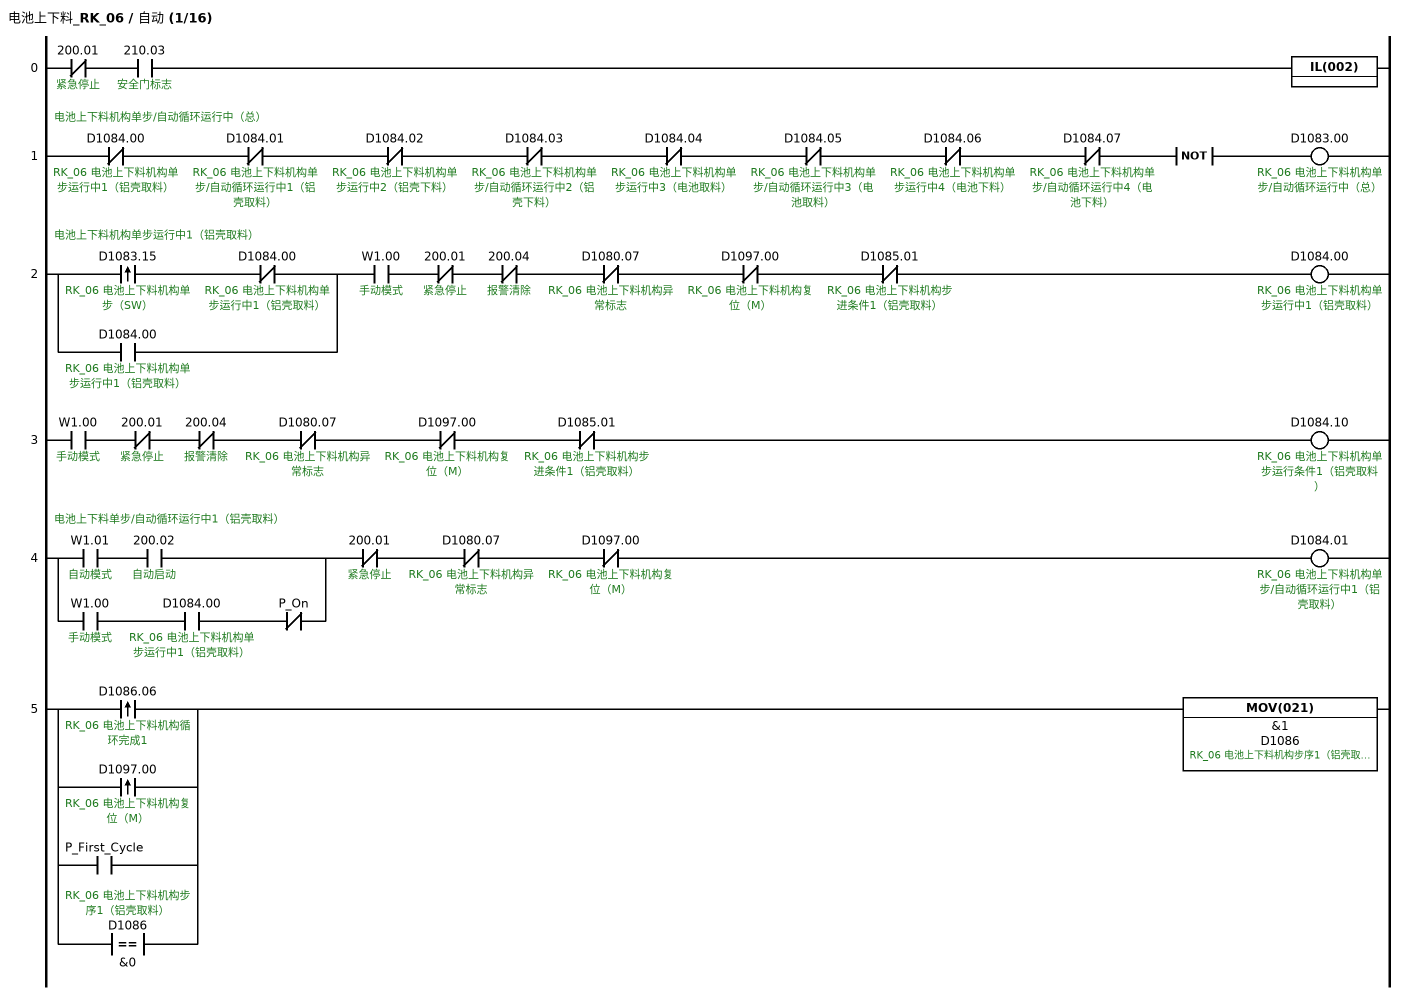
; [picture p528: 电池上下料_RK_06 / 自动, rungs 0-5]
; rung 0
LDNOT 200.01  ; 紧急停止
AND 210.03  ; 安全门标志
IL(002)
; rung 1: 电池上下料机构单步/自动循环运行中（总）
LDNOT D1084.00  ; RK_06 电池上下料机构单步运行中1（铝壳取料）
ANDNOT D1084.01  ; RK_06 电池上下料机构单步/自动循环运行中1（铝壳取料）
ANDNOT D1084.02  ; RK_06 电池上下料机构单步运行中2（铝壳下料）
ANDNOT D1084.03  ; RK_06 电池上下料机构单步/自动循环运行中2（铝壳下料）
ANDNOT D1084.04  ; RK_06 电池上下料机构单步运行中3（电池取料）
ANDNOT D1084.05  ; RK_06 电池上下料机构单步/自动循环运行中3（电池取料）
ANDNOT D1084.06  ; RK_06 电池上下料机构单步运行中4（电池下料）
ANDNOT D1084.07  ; RK_06 电池上下料机构单步/自动循环运行中4（电池下料）
NOT(520)
OUT D1083.00  ; RK_06 电池上下料机构单步/自动循环运行中（总）
; rung 2: 电池上下料机构单步运行中1（铝壳取料）
@LD D1083.15  ; RK_06 电池上下料机构单步（SW）
ANDNOT D1084.00  ; RK_06 电池上下料机构单步运行中1（铝壳取料）
OR D1084.00  ; RK_06 电池上下料机构单步运行中1（铝壳取料）
AND W1.00  ; 手动模式
ANDNOT 200.01  ; 紧急停止
ANDNOT 200.04  ; 报警清除
ANDNOT D1080.07  ; RK_06 电池上下料机构异常标志
ANDNOT D1097.00  ; RK_06 电池上下料机构复位（M）
ANDNOT D1085.01  ; RK_06 电池上下料机构步进条件1（铝壳取料）
OUT D1084.00  ; RK_06 电池上下料机构单步运行中1（铝壳取料）
; rung 3
LD W1.00  ; 手动模式
ANDNOT 200.01  ; 紧急停止
ANDNOT 200.04  ; 报警清除
ANDNOT D1080.07  ; RK_06 电池上下料机构异常标志
ANDNOT D1097.00  ; RK_06 电池上下料机构复位（M）
ANDNOT D1085.01  ; RK_06 电池上下料机构步进条件1（铝壳取料）
OUT D1084.10  ; RK_06 电池上下料机构单步运行条件1（铝壳取料）
; rung 4: 电池上下料单步/自动循环运行中1（铝壳取料）
LD W1.01  ; 自动模式
AND 200.02  ; 自动启动
LD W1.00  ; 手动模式
AND D1084.00  ; RK_06 电池上下料机构单步运行中1（铝壳取料）
ANDNOT P_On
ORLD
ANDNOT 200.01  ; 紧急停止
ANDNOT D1080.07  ; RK_06 电池上下料机构异常标志
ANDNOT D1097.00  ; RK_06 电池上下料机构复位（M）
OUT D1084.01  ; RK_06 电池上下料机构单步/自动循环运行中1（铝壳取料）
; rung 5
@LD D1086.06  ; RK_06 电池上下料机构循环完成1
@OR D1097.00  ; RK_06 电池上下料机构复位（M）
OR P_First_Cycle
OR=(300) D1086 &0  ; RK_06 电池上下料机构步序1（铝壳取料）
MOV(021) &1 D1086  ; RK_06 电池上下料机构步序1（铝壳取料）

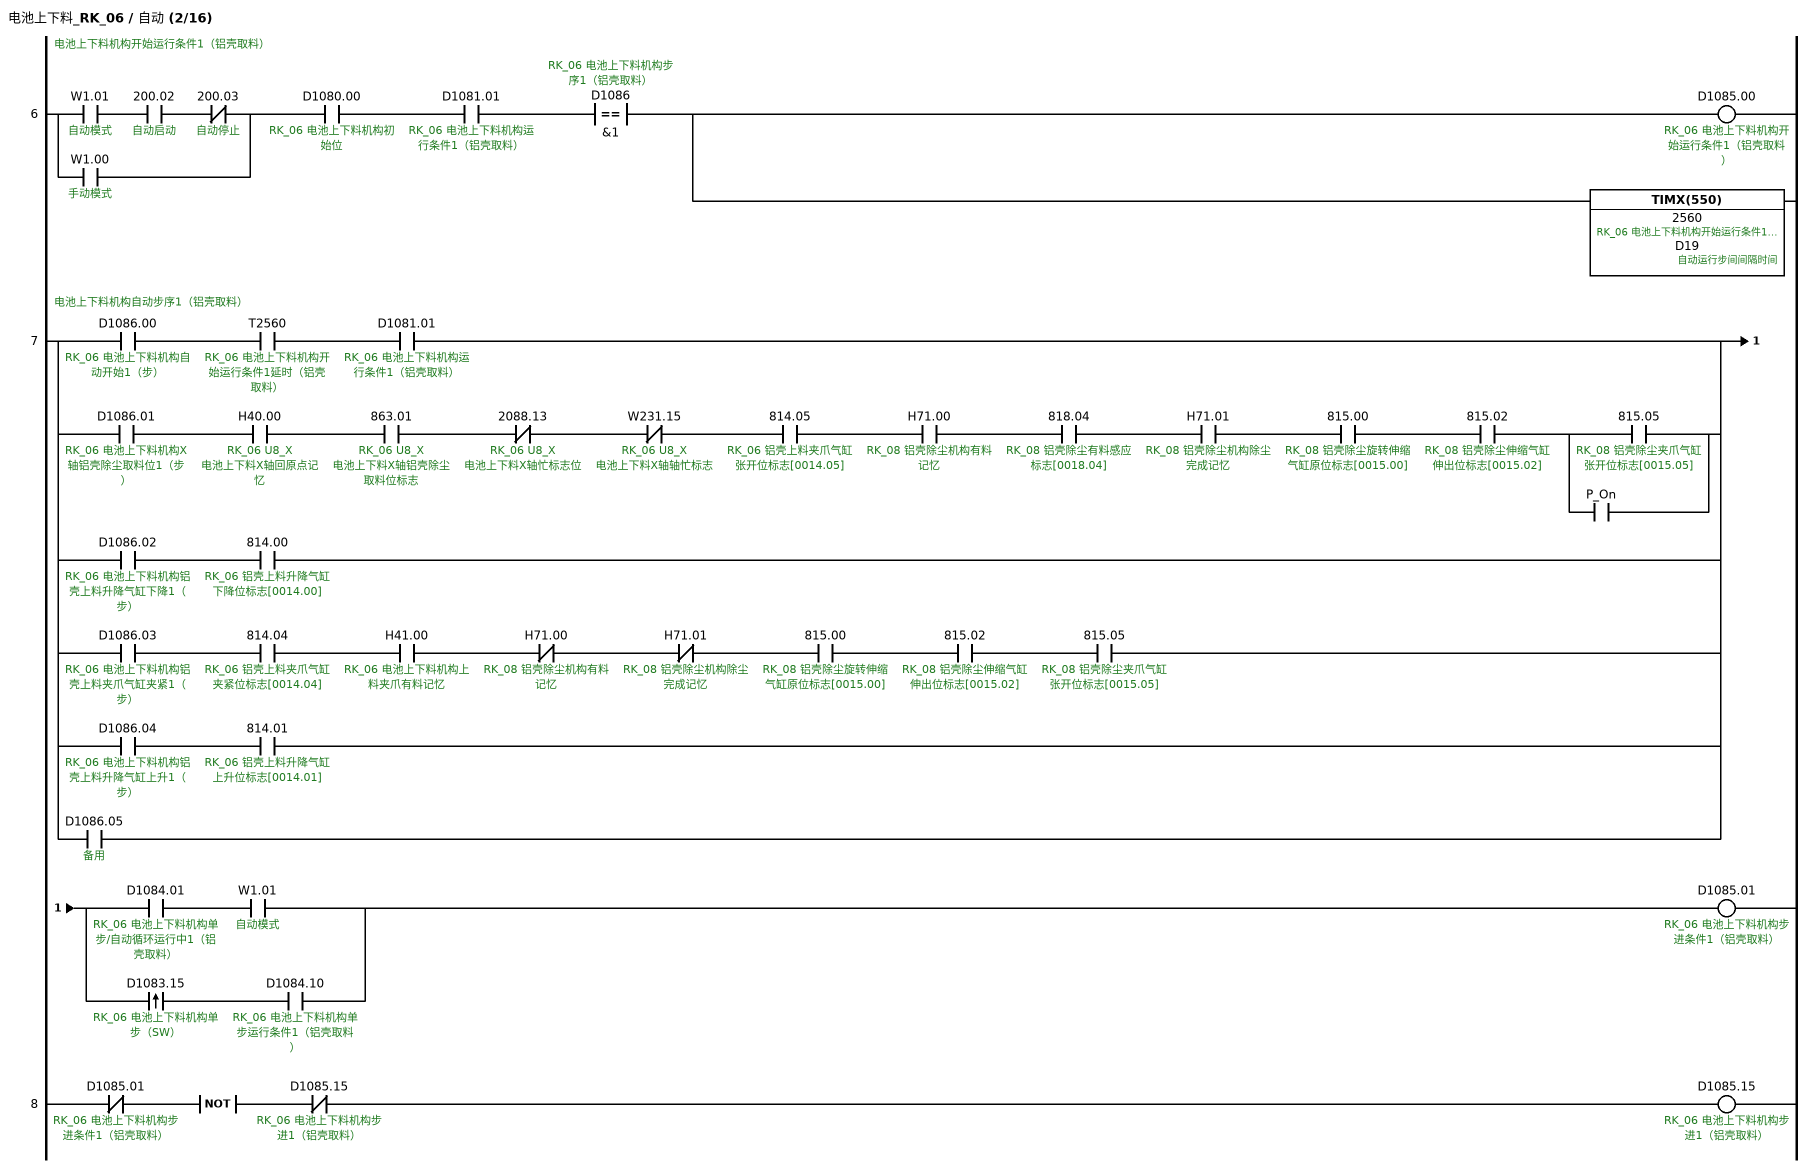
; rung 6: 电池上下料机构开始运行条件1（铝壳取料）
LD W1.01  ; 自动模式
AND 200.02  ; 自动启动
ANDNOT 200.03  ; 自动停止
OR W1.00  ; 手动模式
AND D1080.00  ; RK_06 电池上下料机构初始位
AND D1081.01  ; RK_06 电池上下料机构运行条件1（铝壳取料）
AND=(300) D1086 &1  ; RK_06 电池上下料机构步序1（铝壳取料）
OUT D1085.00  ; RK_06 电池上下料机构开始运行条件1（铝壳取料）
TIMX(550) 2560 D19  ; 自动运行步间间隔时间, RK_06 电池上下料机构开始运行条件1延时（铝壳取料）
; rung 7: 电池上下料机构自动步序1（铝壳取料）
LD D1086.00  ; RK_06 电池上下料机构自动开始1（步）
AND T2560  ; RK_06 电池上下料机构开始运行条件1延时（铝壳取料）
AND D1081.01  ; RK_06 电池上下料机构运行条件1（铝壳取料）
LD D1086.01  ; RK_06 电池上下料机构X轴铝壳除尘取料位1（步）
AND H40.00  ; RK_06 U8_X 电池上下料X轴回原点记忆
AND 863.01  ; RK_06 U8_X 电池上下料X轴铝壳除尘取料位标志
ANDNOT 2088.13  ; RK_06 U8_X 电池上下料X轴忙标志位
ANDNOT W231.15  ; RK_06 U8_X 电池上下料X轴轴忙标志
AND 814.05  ; RK_06 铝壳上料夹爪气缸张开位标志[0014.05]
AND H71.00  ; RK_08 铝壳除尘机构有料记忆
AND 818.04  ; RK_08 铝壳除尘有料感应标志[0018.04]
AND H71.01  ; RK_08 铝壳除尘机构除尘完成记忆
AND 815.00  ; RK_08 铝壳除尘旋转伸缩气缸原位标志[0015.00]
AND 815.02  ; RK_08 铝壳除尘伸缩气缸伸出位标志[0015.02]
LD 815.05  ; RK_08 铝壳除尘夹爪气缸张开位标志[0015.05]
OR P_On
ANDLD
ORLD
LD D1086.02  ; RK_06 电池上下料机构铝壳上料升降气缸下降1（步）
AND 814.00  ; RK_06 铝壳上料升降气缸下降位标志[0014.00]
ORLD
LD D1086.03  ; RK_06 电池上下料机构铝壳上料夹爪气缸夹紧1（步）
AND 814.04  ; RK_06 铝壳上料夹爪气缸夹紧位标志[0014.04]
AND H41.00  ; RK_06 电池上下料机构上料夹爪有料记忆
ANDNOT H71.00  ; RK_08 铝壳除尘机构有料记忆
ANDNOT H71.01  ; RK_08 铝壳除尘机构除尘完成记忆
AND 815.00  ; RK_08 铝壳除尘旋转伸缩气缸原位标志[0015.00]
AND 815.02  ; RK_08 铝壳除尘伸缩气缸伸出位标志[0015.02]
AND 815.05  ; RK_08 铝壳除尘夹爪气缸张开位标志[0015.05]
ORLD
LD D1086.04  ; RK_06 电池上下料机构铝壳上料升降气缸上升1（步）
AND 814.01  ; RK_06 铝壳上料升降气缸上升位标志[0014.01]
ORLD
OR D1086.05  ; 备用
LD D1084.01  ; RK_06 电池上下料机构单步/自动循环运行中1（铝壳取料）
AND W1.01  ; 自动模式
@LD D1083.15  ; RK_06 电池上下料机构单步（SW）
AND D1084.10  ; RK_06 电池上下料机构单步运行条件1（铝壳取料）
ORLD
ANDLD
OUT D1085.01  ; RK_06 电池上下料机构步进条件1（铝壳取料）
; rung 8
LDNOT D1085.01  ; RK_06 电池上下料机构步进条件1（铝壳取料）
NOT(520)
ANDNOT D1085.15  ; RK_06 电池上下料机构步进1（铝壳取料）
OUT D1085.15  ; RK_06 电池上下料机构步进1（铝壳取料）

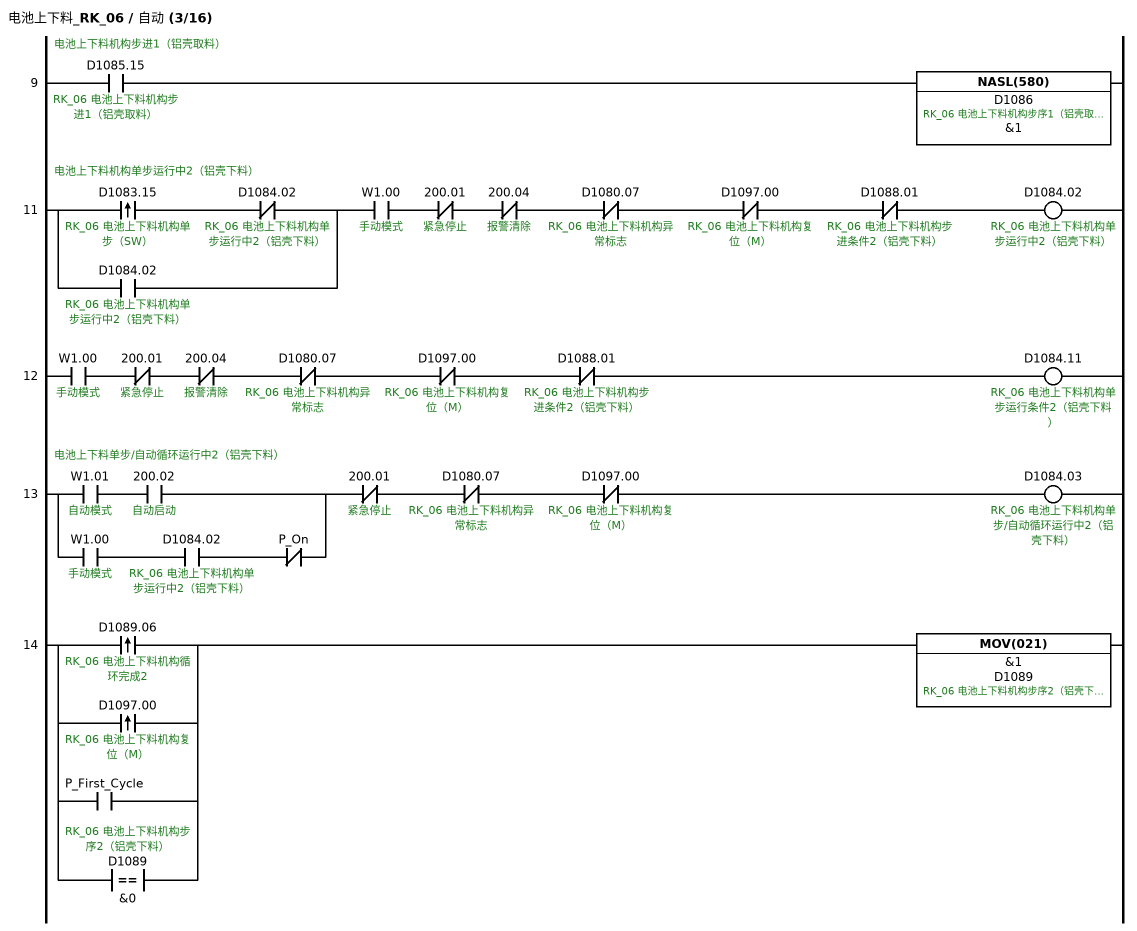
; rung 9: 电池上下料机构步进1（铝壳取料）
LD D1085.15  ; RK_06 电池上下料机构步进1（铝壳取料）
NASL(580) D1086 &1  ; RK_06 电池上下料机构步序1（铝壳取料）
; rung 10: 电池上下料机构步序跳转1（铝壳取料）
; rung 11: 电池上下料机构单步运行中2（铝壳下料）
@LD D1083.15  ; RK_06 电池上下料机构单步（SW）
ANDNOT D1084.02  ; RK_06 电池上下料机构单步运行中2（铝壳下料）
OR D1084.02  ; RK_06 电池上下料机构单步运行中2（铝壳下料）
AND W1.00  ; 手动模式
ANDNOT 200.01  ; 紧急停止
ANDNOT 200.04  ; 报警清除
ANDNOT D1080.07  ; RK_06 电池上下料机构异常标志
ANDNOT D1097.00  ; RK_06 电池上下料机构复位（M）
ANDNOT D1088.01  ; RK_06 电池上下料机构步进条件2（铝壳下料）
OUT D1084.02  ; RK_06 电池上下料机构单步运行中2（铝壳下料）
; rung 12
LD W1.00  ; 手动模式
ANDNOT 200.01  ; 紧急停止
ANDNOT 200.04  ; 报警清除
ANDNOT D1080.07  ; RK_06 电池上下料机构异常标志
ANDNOT D1097.00  ; RK_06 电池上下料机构复位（M）
ANDNOT D1088.01  ; RK_06 电池上下料机构步进条件2（铝壳下料）
OUT D1084.11  ; RK_06 电池上下料机构单步运行条件2（铝壳下料）
; rung 13: 电池上下料单步/自动循环运行中2（铝壳下料）
LD W1.01  ; 自动模式
AND 200.02  ; 自动启动
LD W1.00  ; 手动模式
AND D1084.02  ; RK_06 电池上下料机构单步运行中2（铝壳下料）
ANDNOT P_On
ORLD
ANDNOT 200.01  ; 紧急停止
ANDNOT D1080.07  ; RK_06 电池上下料机构异常标志
ANDNOT D1097.00  ; RK_06 电池上下料机构复位（M）
OUT D1084.03  ; RK_06 电池上下料机构单步/自动循环运行中2（铝壳下料）
; rung 14
@LD D1089.06  ; RK_06 电池上下料机构循环完成2
@OR D1097.00  ; RK_06 电池上下料机构复位（M）
OR P_First_Cycle
OR=(300) D1089 &0  ; RK_06 电池上下料机构步序2（铝壳下料）
MOV(021) &1 D1089  ; RK_06 电池上下料机构步序2（铝壳下料）

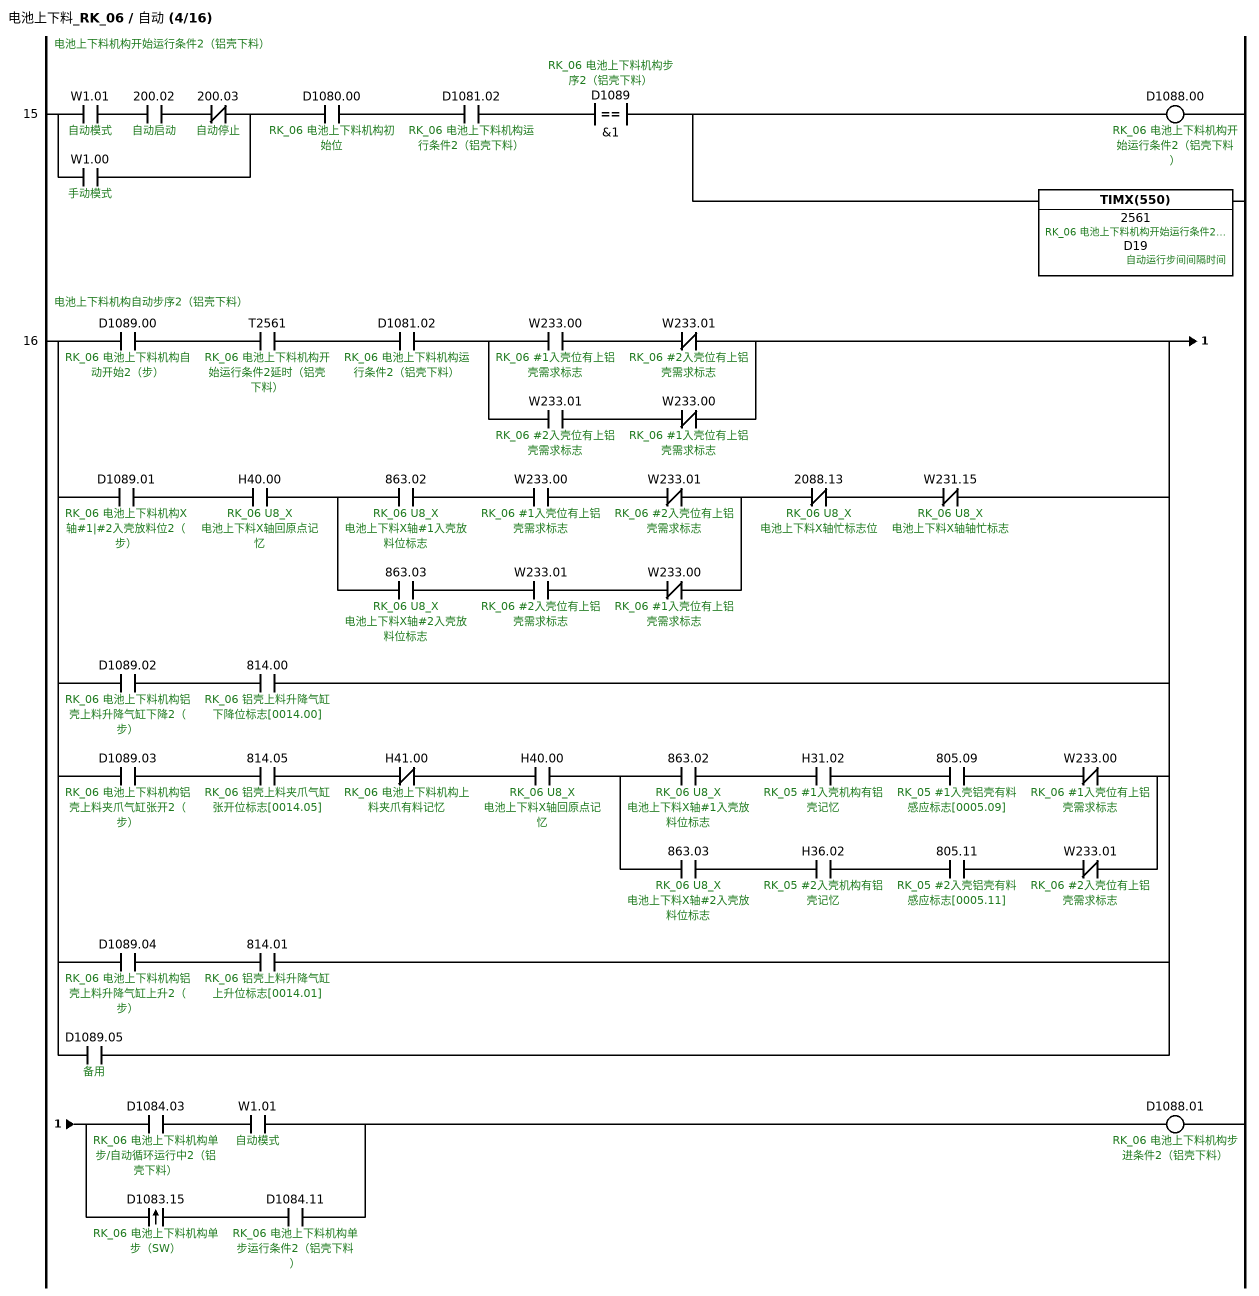
; rung 15: 电池上下料机构开始运行条件2（铝壳下料）
LD W1.01  ; 自动模式
AND 200.02  ; 自动启动
ANDNOT 200.03  ; 自动停止
OR W1.00  ; 手动模式
AND D1080.00  ; RK_06 电池上下料机构初始位
AND D1081.02  ; RK_06 电池上下料机构运行条件2（铝壳下料）
AND=(300) D1089 &1  ; RK_06 电池上下料机构步序2（铝壳下料）
OUT D1088.00  ; RK_06 电池上下料机构开始运行条件2（铝壳下料）
TIMX(550) 2561 D19  ; 自动运行步间间隔时间, RK_06 电池上下料机构开始运行条件2延时（铝壳下料）
; rung 16: 电池上下料机构自动步序2（铝壳下料）
LD D1089.00  ; RK_06 电池上下料机构自动开始2（步）
AND T2561  ; RK_06 电池上下料机构开始运行条件2延时（铝壳下料）
AND D1081.02  ; RK_06 电池上下料机构运行条件2（铝壳下料）
LD W233.00  ; RK_06 #1入壳位有上铝壳需求标志
ANDNOT W233.01  ; RK_06 #2入壳位有上铝壳需求标志
LD W233.01  ; RK_06 #2入壳位有上铝壳需求标志
ANDNOT W233.00  ; RK_06 #1入壳位有上铝壳需求标志
ORLD
ANDLD
LD D1089.01  ; RK_06 电池上下料机构X轴#1|#2入壳放料位2（步）
AND H40.00  ; RK_06 U8_X 电池上下料X轴回原点记忆
LD 863.02  ; RK_06 U8_X 电池上下料X轴#1入壳放料位标志
AND W233.00  ; RK_06 #1入壳位有上铝壳需求标志
ANDNOT W233.01  ; RK_06 #2入壳位有上铝壳需求标志
LD 863.03  ; RK_06 U8_X 电池上下料X轴#2入壳放料位标志
AND W233.01  ; RK_06 #2入壳位有上铝壳需求标志
ANDNOT W233.00  ; RK_06 #1入壳位有上铝壳需求标志
ORLD
ANDLD
ANDNOT 2088.13  ; RK_06 U8_X 电池上下料X轴忙标志位
ANDNOT W231.15  ; RK_06 U8_X 电池上下料X轴轴忙标志
ORLD
LD D1089.02  ; RK_06 电池上下料机构铝壳上料升降气缸下降2（步）
AND 814.00  ; RK_06 铝壳上料升降气缸下降位标志[0014.00]
ORLD
LD D1089.03  ; RK_06 电池上下料机构铝壳上料夹爪气缸张开2（步）
AND 814.05  ; RK_06 铝壳上料夹爪气缸张开位标志[0014.05]
ANDNOT H41.00  ; RK_06 电池上下料机构上料夹爪有料记忆
AND H40.00  ; RK_06 U8_X 电池上下料X轴回原点记忆
LD 863.02  ; RK_06 U8_X 电池上下料X轴#1入壳放料位标志
AND H31.02  ; RK_05 #1入壳机构有铝壳记忆
AND 805.09  ; RK_05 #1入壳铝壳有料感应标志[0005.09]
ANDNOT W233.00  ; RK_06 #1入壳位有上铝壳需求标志
LD 863.03  ; RK_06 U8_X 电池上下料X轴#2入壳放料位标志
AND H36.02  ; RK_05 #2入壳机构有铝壳记忆
AND 805.11  ; RK_05 #2入壳铝壳有料感应标志[0005.11]
ANDNOT W233.01  ; RK_06 #2入壳位有上铝壳需求标志
ORLD
ANDLD
ORLD
LD D1089.04  ; RK_06 电池上下料机构铝壳上料升降气缸上升2（步）
AND 814.01  ; RK_06 铝壳上料升降气缸上升位标志[0014.01]
ORLD
OR D1089.05  ; 备用
LD D1084.03  ; RK_06 电池上下料机构单步/自动循环运行中2（铝壳下料）
AND W1.01  ; 自动模式
@LD D1083.15  ; RK_06 电池上下料机构单步（SW）
AND D1084.11  ; RK_06 电池上下料机构单步运行条件2（铝壳下料）
ORLD
ANDLD
OUT D1088.01  ; RK_06 电池上下料机构步进条件2（铝壳下料）

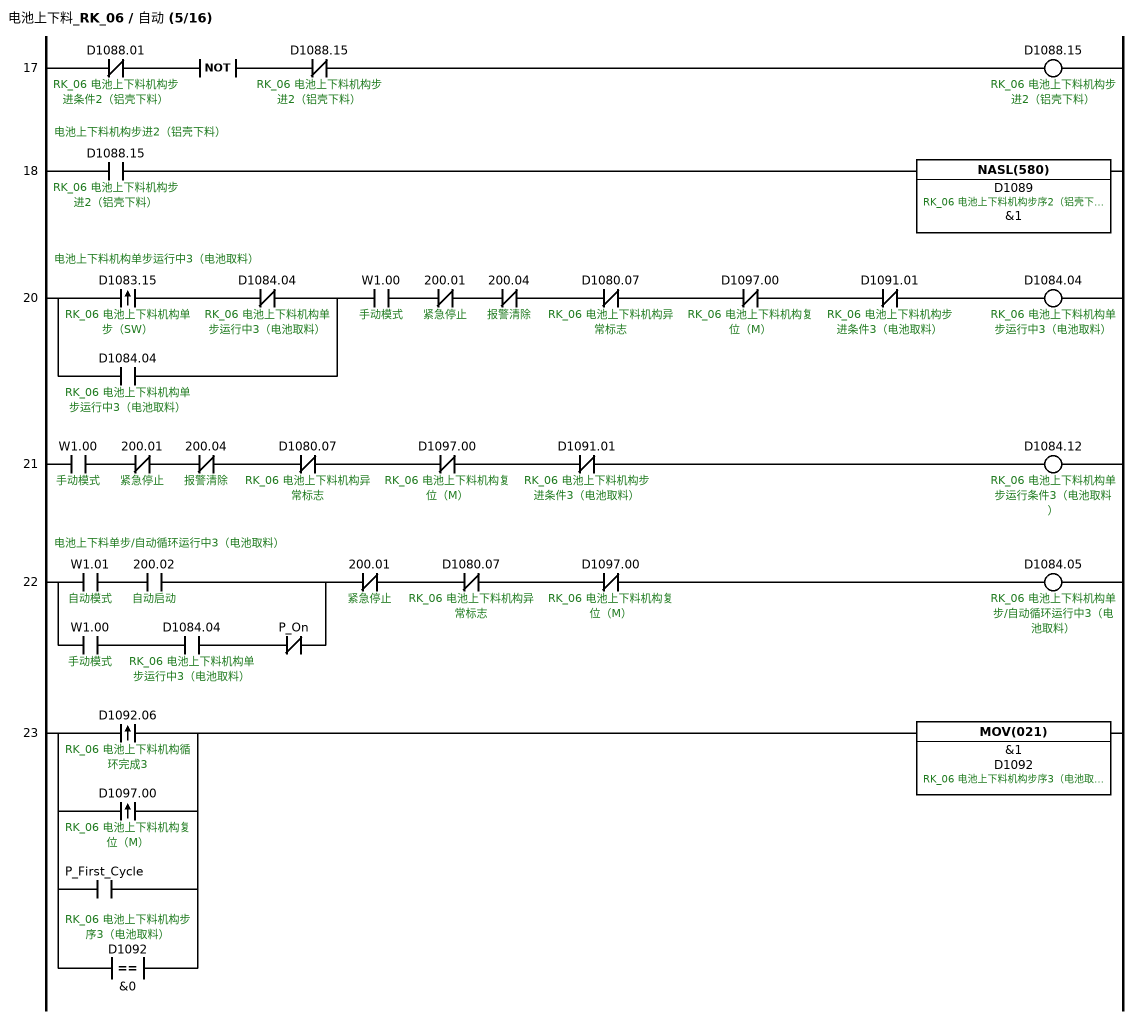
; rung 17
LDNOT D1088.01  ; RK_06 电池上下料机构步进条件2（铝壳下料）
NOT(520)
ANDNOT D1088.15  ; RK_06 电池上下料机构步进2（铝壳下料）
OUT D1088.15  ; RK_06 电池上下料机构步进2（铝壳下料）
; rung 18: 电池上下料机构步进2（铝壳下料）
LD D1088.15  ; RK_06 电池上下料机构步进2（铝壳下料）
NASL(580) D1089 &1  ; RK_06 电池上下料机构步序2（铝壳下料）
; rung 19: 电池上下料机构步序跳转2（铝壳下料）
; rung 20: 电池上下料机构单步运行中3（电池取料）
@LD D1083.15  ; RK_06 电池上下料机构单步（SW）
ANDNOT D1084.04  ; RK_06 电池上下料机构单步运行中3（电池取料）
OR D1084.04  ; RK_06 电池上下料机构单步运行中3（电池取料）
AND W1.00  ; 手动模式
ANDNOT 200.01  ; 紧急停止
ANDNOT 200.04  ; 报警清除
ANDNOT D1080.07  ; RK_06 电池上下料机构异常标志
ANDNOT D1097.00  ; RK_06 电池上下料机构复位（M）
ANDNOT D1091.01  ; RK_06 电池上下料机构步进条件3（电池取料）
OUT D1084.04  ; RK_06 电池上下料机构单步运行中3（电池取料）
; rung 21
LD W1.00  ; 手动模式
ANDNOT 200.01  ; 紧急停止
ANDNOT 200.04  ; 报警清除
ANDNOT D1080.07  ; RK_06 电池上下料机构异常标志
ANDNOT D1097.00  ; RK_06 电池上下料机构复位（M）
ANDNOT D1091.01  ; RK_06 电池上下料机构步进条件3（电池取料）
OUT D1084.12  ; RK_06 电池上下料机构单步运行条件3（电池取料）
; rung 22: 电池上下料单步/自动循环运行中3（电池取料）
LD W1.01  ; 自动模式
AND 200.02  ; 自动启动
LD W1.00  ; 手动模式
AND D1084.04  ; RK_06 电池上下料机构单步运行中3（电池取料）
ANDNOT P_On
ORLD
ANDNOT 200.01  ; 紧急停止
ANDNOT D1080.07  ; RK_06 电池上下料机构异常标志
ANDNOT D1097.00  ; RK_06 电池上下料机构复位（M）
OUT D1084.05  ; RK_06 电池上下料机构单步/自动循环运行中3（电池取料）
; rung 23
@LD D1092.06  ; RK_06 电池上下料机构循环完成3
@OR D1097.00  ; RK_06 电池上下料机构复位（M）
OR P_First_Cycle
OR=(300) D1092 &0  ; RK_06 电池上下料机构步序3（电池取料）
MOV(021) &1 D1092  ; RK_06 电池上下料机构步序3（电池取料）

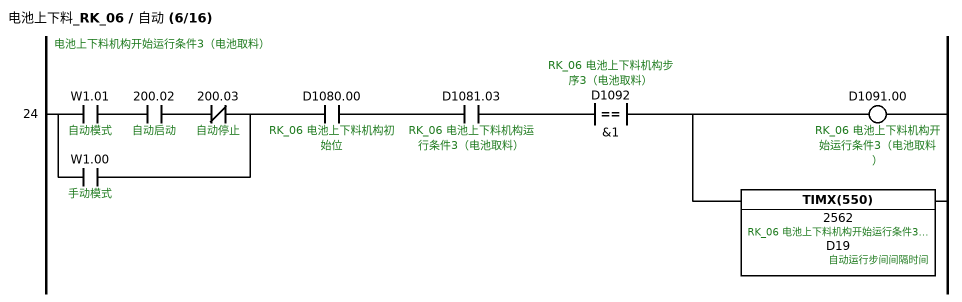
; rung 24: 电池上下料机构开始运行条件3（电池取料）
LD W1.01  ; 自动模式
AND 200.02  ; 自动启动
ANDNOT 200.03  ; 自动停止
OR W1.00  ; 手动模式
AND D1080.00  ; RK_06 电池上下料机构初始位
AND D1081.03  ; RK_06 电池上下料机构运行条件3（电池取料）
AND=(300) D1092 &1  ; RK_06 电池上下料机构步序3（电池取料）
OUT D1091.00  ; RK_06 电池上下料机构开始运行条件3（电池取料）
TIMX(550) 2562 D19  ; 自动运行步间间隔时间, RK_06 电池上下料机构开始运行条件3延时（电池取料）

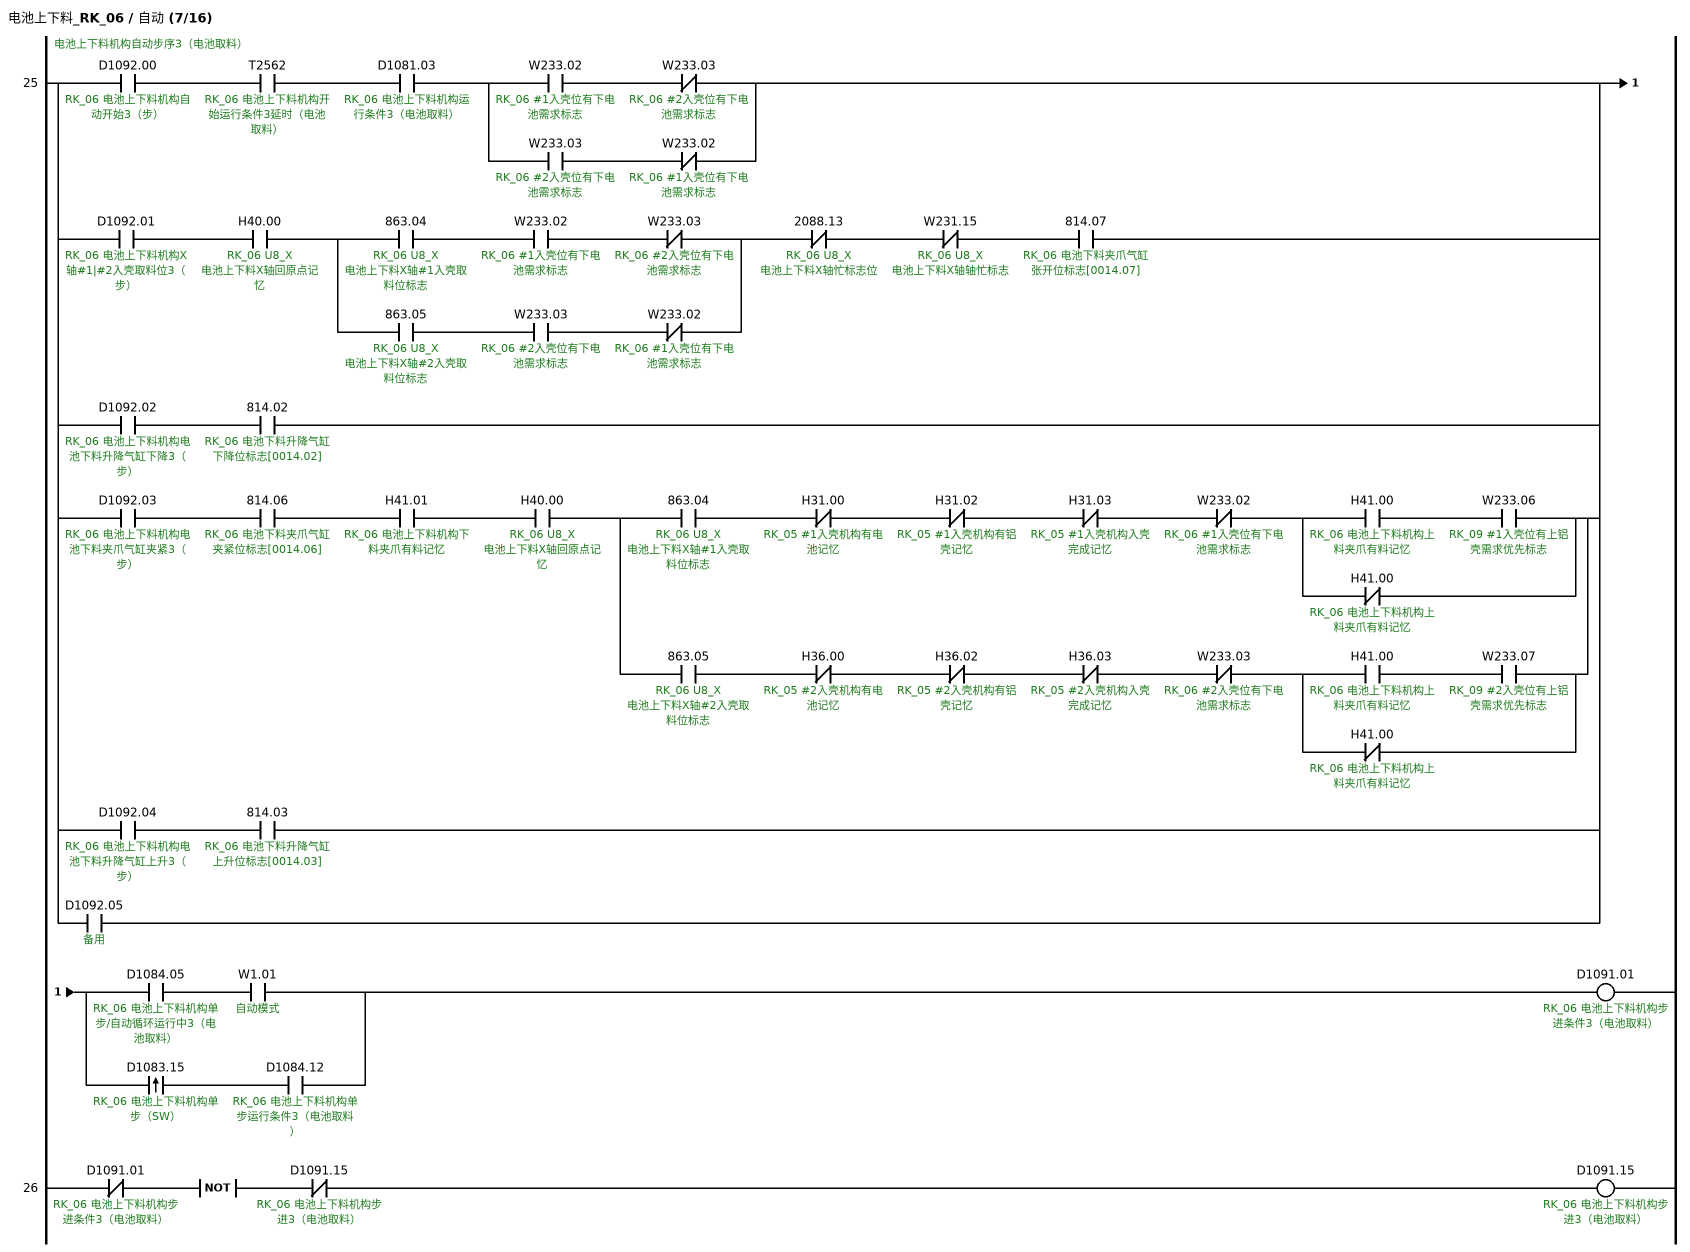
; rung 25: 电池上下料机构自动步序3（电池取料）
LD D1092.00  ; RK_06 电池上下料机构自动开始3（步）
AND T2562  ; RK_06 电池上下料机构开始运行条件3延时（电池取料）
AND D1081.03  ; RK_06 电池上下料机构运行条件3（电池取料）
LD W233.02  ; RK_06 #1入壳位有下电池需求标志
ANDNOT W233.03  ; RK_06 #2入壳位有下电池需求标志
LD W233.03  ; RK_06 #2入壳位有下电池需求标志
ANDNOT W233.02  ; RK_06 #1入壳位有下电池需求标志
ORLD
ANDLD
LD D1092.01  ; RK_06 电池上下料机构X轴#1|#2入壳取料位3（步）
AND H40.00  ; RK_06 U8_X 电池上下料X轴回原点记忆
LD 863.04  ; RK_06 U8_X 电池上下料X轴#1入壳取料位标志
AND W233.02  ; RK_06 #1入壳位有下电池需求标志
ANDNOT W233.03  ; RK_06 #2入壳位有下电池需求标志
LD 863.05  ; RK_06 U8_X 电池上下料X轴#2入壳取料位标志
AND W233.03  ; RK_06 #2入壳位有下电池需求标志
ANDNOT W233.02  ; RK_06 #1入壳位有下电池需求标志
ORLD
ANDLD
ANDNOT 2088.13  ; RK_06 U8_X 电池上下料X轴忙标志位
ANDNOT W231.15  ; RK_06 U8_X 电池上下料X轴轴忙标志
AND 814.07  ; RK_06 电池下料夹爪气缸张开位标志[0014.07]
ORLD
LD D1092.02  ; RK_06 电池上下料机构电池下料升降气缸下降3（步）
AND 814.02  ; RK_06 电池下料升降气缸下降位标志[0014.02]
ORLD
LD D1092.03  ; RK_06 电池上下料机构电池下料夹爪气缸夹紧3（步）
AND 814.06  ; RK_06 电池下料夹爪气缸夹紧位标志[0014.06]
AND H41.01  ; RK_06 电池上下料机构下料夹爪有料记忆
AND H40.00  ; RK_06 U8_X 电池上下料X轴回原点记忆
LD 863.04  ; RK_06 U8_X 电池上下料X轴#1入壳取料位标志
ANDNOT H31.00  ; RK_05 #1入壳机构有电池记忆
ANDNOT H31.02  ; RK_05 #1入壳机构有铝壳记忆
ANDNOT H31.03  ; RK_05 #1入壳机构入壳完成记忆
ANDNOT W233.02  ; RK_06 #1入壳位有下电池需求标志
LD H41.00  ; RK_06 电池上下料机构上料夹爪有料记忆
AND W233.06  ; RK_09 #1入壳位有上铝壳需求优先标志
ORNOT H41.00  ; RK_06 电池上下料机构上料夹爪有料记忆
ANDLD
LD 863.05  ; RK_06 U8_X 电池上下料X轴#2入壳取料位标志
ANDNOT H36.00  ; RK_05 #2入壳机构有电池记忆
ANDNOT H36.02  ; RK_05 #2入壳机构有铝壳记忆
ANDNOT H36.03  ; RK_05 #2入壳机构入壳完成记忆
ANDNOT W233.03  ; RK_06 #2入壳位有下电池需求标志
LD H41.00  ; RK_06 电池上下料机构上料夹爪有料记忆
AND W233.07  ; RK_09 #2入壳位有上铝壳需求优先标志
ORNOT H41.00  ; RK_06 电池上下料机构上料夹爪有料记忆
ANDLD
ORLD
ANDLD
ORLD
LD D1092.04  ; RK_06 电池上下料机构电池下料升降气缸上升3（步）
AND 814.03  ; RK_06 电池下料升降气缸上升位标志[0014.03]
ORLD
OR D1092.05  ; 备用
LD D1084.05  ; RK_06 电池上下料机构单步/自动循环运行中3（电池取料）
AND W1.01  ; 自动模式
@LD D1083.15  ; RK_06 电池上下料机构单步（SW）
AND D1084.12  ; RK_06 电池上下料机构单步运行条件3（电池取料）
ORLD
ANDLD
OUT D1091.01  ; RK_06 电池上下料机构步进条件3（电池取料）
; rung 26
LDNOT D1091.01  ; RK_06 电池上下料机构步进条件3（电池取料）
NOT(520)
ANDNOT D1091.15  ; RK_06 电池上下料机构步进3（电池取料）
OUT D1091.15  ; RK_06 电池上下料机构步进3（电池取料）

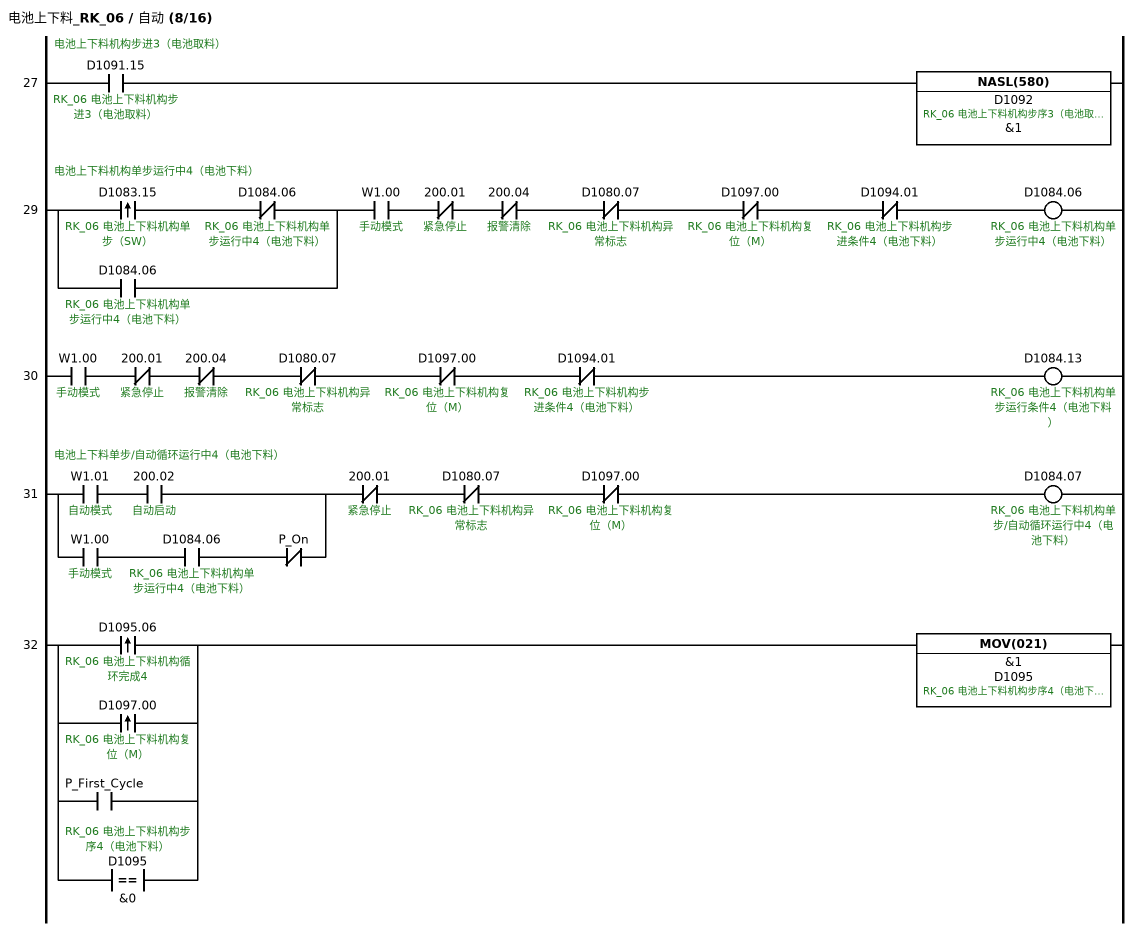
; rung 27: 电池上下料机构步进3（电池取料）
LD D1091.15  ; RK_06 电池上下料机构步进3（电池取料）
NASL(580) D1092 &1  ; RK_06 电池上下料机构步序3（电池取料）
; rung 28: 电池上下料机构步序跳转3（电池取料）
; rung 29: 电池上下料机构单步运行中4（电池下料）
@LD D1083.15  ; RK_06 电池上下料机构单步（SW）
ANDNOT D1084.06  ; RK_06 电池上下料机构单步运行中4（电池下料）
OR D1084.06  ; RK_06 电池上下料机构单步运行中4（电池下料）
AND W1.00  ; 手动模式
ANDNOT 200.01  ; 紧急停止
ANDNOT 200.04  ; 报警清除
ANDNOT D1080.07  ; RK_06 电池上下料机构异常标志
ANDNOT D1097.00  ; RK_06 电池上下料机构复位（M）
ANDNOT D1094.01  ; RK_06 电池上下料机构步进条件4（电池下料）
OUT D1084.06  ; RK_06 电池上下料机构单步运行中4（电池下料）
; rung 30
LD W1.00  ; 手动模式
ANDNOT 200.01  ; 紧急停止
ANDNOT 200.04  ; 报警清除
ANDNOT D1080.07  ; RK_06 电池上下料机构异常标志
ANDNOT D1097.00  ; RK_06 电池上下料机构复位（M）
ANDNOT D1094.01  ; RK_06 电池上下料机构步进条件4（电池下料）
OUT D1084.13  ; RK_06 电池上下料机构单步运行条件4（电池下料）
; rung 31: 电池上下料单步/自动循环运行中4（电池下料）
LD W1.01  ; 自动模式
AND 200.02  ; 自动启动
LD W1.00  ; 手动模式
AND D1084.06  ; RK_06 电池上下料机构单步运行中4（电池下料）
ANDNOT P_On
ORLD
ANDNOT 200.01  ; 紧急停止
ANDNOT D1080.07  ; RK_06 电池上下料机构异常标志
ANDNOT D1097.00  ; RK_06 电池上下料机构复位（M）
OUT D1084.07  ; RK_06 电池上下料机构单步/自动循环运行中4（电池下料）
; rung 32
@LD D1095.06  ; RK_06 电池上下料机构循环完成4
@OR D1097.00  ; RK_06 电池上下料机构复位（M）
OR P_First_Cycle
OR=(300) D1095 &0  ; RK_06 电池上下料机构步序4（电池下料）
MOV(021) &1 D1095  ; RK_06 电池上下料机构步序4（电池下料）

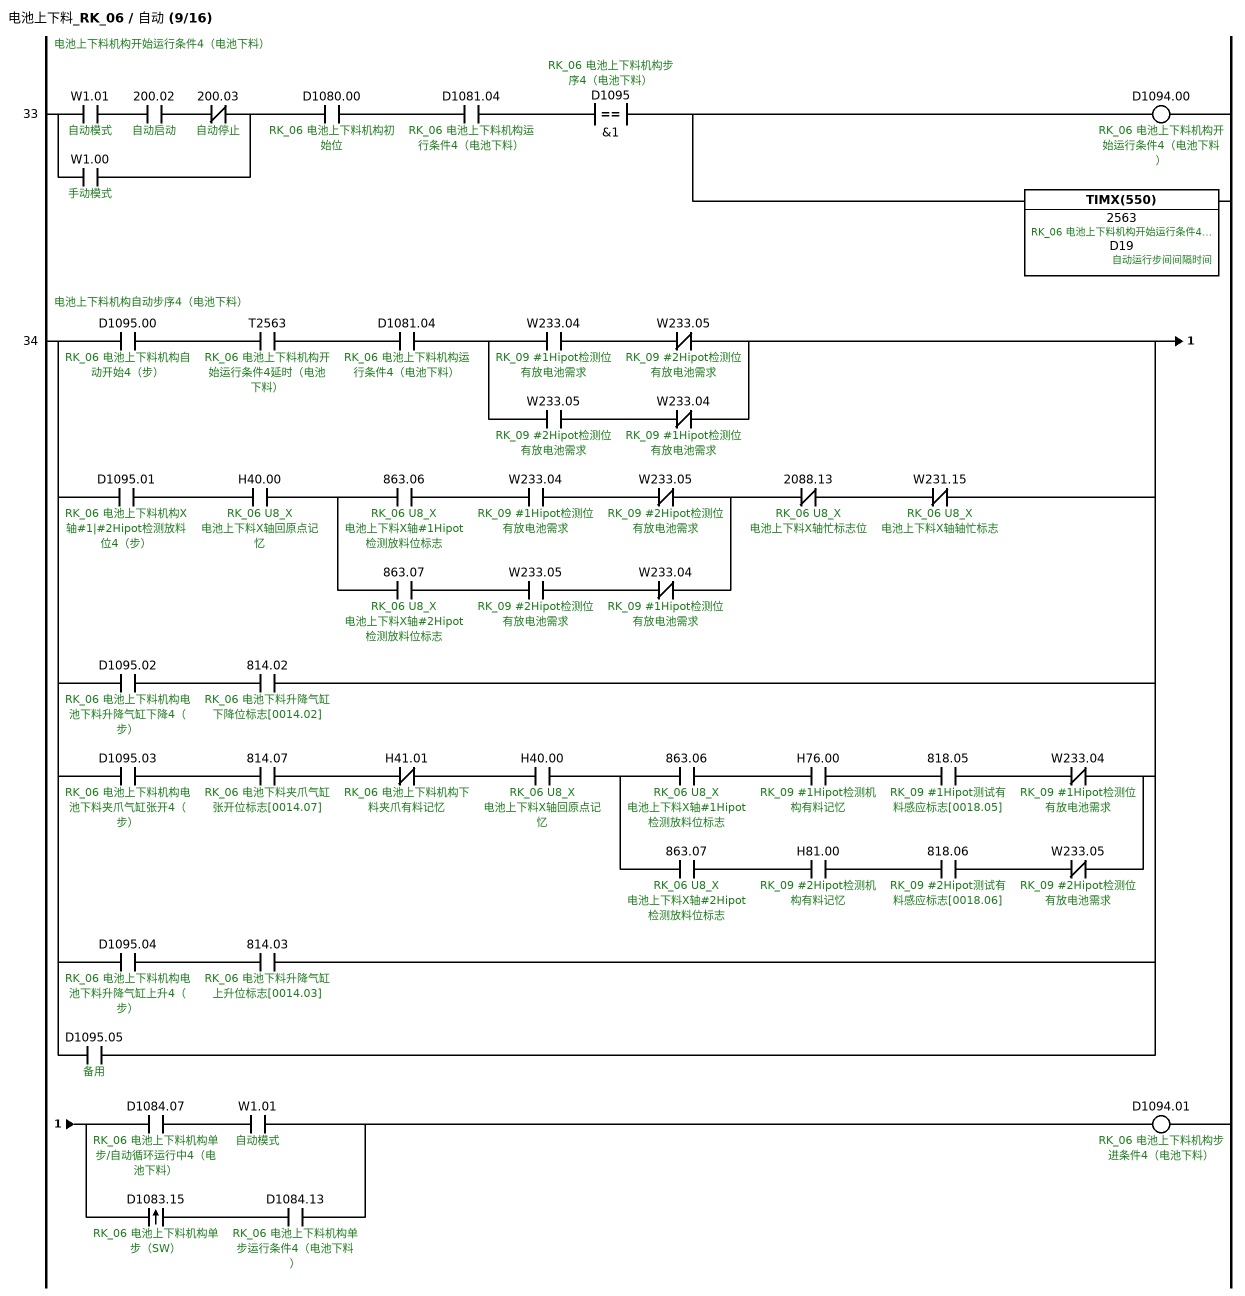
; rung 33: 电池上下料机构开始运行条件4（电池下料）
LD W1.01  ; 自动模式
AND 200.02  ; 自动启动
ANDNOT 200.03  ; 自动停止
OR W1.00  ; 手动模式
AND D1080.00  ; RK_06 电池上下料机构初始位
AND D1081.04  ; RK_06 电池上下料机构运行条件4（电池下料）
AND=(300) D1095 &1  ; RK_06 电池上下料机构步序4（电池下料）
OUT D1094.00  ; RK_06 电池上下料机构开始运行条件4（电池下料）
TIMX(550) 2563 D19  ; 自动运行步间间隔时间, RK_06 电池上下料机构开始运行条件4延时（电池下料）
; rung 34: 电池上下料机构自动步序4（电池下料）
LD D1095.00  ; RK_06 电池上下料机构自动开始4（步）
AND T2563  ; RK_06 电池上下料机构开始运行条件4延时（电池下料）
AND D1081.04  ; RK_06 电池上下料机构运行条件4（电池下料）
LD W233.04  ; RK_09 #1Hipot检测位有放电池需求
ANDNOT W233.05  ; RK_09 #2Hipot检测位有放电池需求
LD W233.05  ; RK_09 #2Hipot检测位有放电池需求
ANDNOT W233.04  ; RK_09 #1Hipot检测位有放电池需求
ORLD
ANDLD
LD D1095.01  ; RK_06 电池上下料机构X轴#1|#2Hipot检测放料位4（步）
AND H40.00  ; RK_06 U8_X 电池上下料X轴回原点记忆
LD 863.06  ; RK_06 U8_X 电池上下料X轴#1Hipot检测放料位标志
AND W233.04  ; RK_09 #1Hipot检测位有放电池需求
ANDNOT W233.05  ; RK_09 #2Hipot检测位有放电池需求
LD 863.07  ; RK_06 U8_X 电池上下料X轴#2Hipot检测放料位标志
AND W233.05  ; RK_09 #2Hipot检测位有放电池需求
ANDNOT W233.04  ; RK_09 #1Hipot检测位有放电池需求
ORLD
ANDLD
ANDNOT 2088.13  ; RK_06 U8_X 电池上下料X轴忙标志位
ANDNOT W231.15  ; RK_06 U8_X 电池上下料X轴轴忙标志
ORLD
LD D1095.02  ; RK_06 电池上下料机构电池下料升降气缸下降4（步）
AND 814.02  ; RK_06 电池下料升降气缸下降位标志[0014.02]
ORLD
LD D1095.03  ; RK_06 电池上下料机构电池下料夹爪气缸张开4（步）
AND 814.07  ; RK_06 电池下料夹爪气缸张开位标志[0014.07]
ANDNOT H41.01  ; RK_06 电池上下料机构下料夹爪有料记忆
AND H40.00  ; RK_06 U8_X 电池上下料X轴回原点记忆
LD 863.06  ; RK_06 U8_X 电池上下料X轴#1Hipot检测放料位标志
AND H76.00  ; RK_09 #1Hipot检测机构有料记忆
AND 818.05  ; RK_09 #1Hipot测试有料感应标志[0018.05]
ANDNOT W233.04  ; RK_09 #1Hipot检测位有放电池需求
LD 863.07  ; RK_06 U8_X 电池上下料X轴#2Hipot检测放料位标志
AND H81.00  ; RK_09 #2Hipot检测机构有料记忆
AND 818.06  ; RK_09 #2Hipot测试有料感应标志[0018.06]
ANDNOT W233.05  ; RK_09 #2Hipot检测位有放电池需求
ORLD
ANDLD
ORLD
LD D1095.04  ; RK_06 电池上下料机构电池下料升降气缸上升4（步）
AND 814.03  ; RK_06 电池下料升降气缸上升位标志[0014.03]
ORLD
OR D1095.05  ; 备用
LD D1084.07  ; RK_06 电池上下料机构单步/自动循环运行中4（电池下料）
AND W1.01  ; 自动模式
@LD D1083.15  ; RK_06 电池上下料机构单步（SW）
AND D1084.13  ; RK_06 电池上下料机构单步运行条件4（电池下料）
ORLD
ANDLD
OUT D1094.01  ; RK_06 电池上下料机构步进条件4（电池下料）

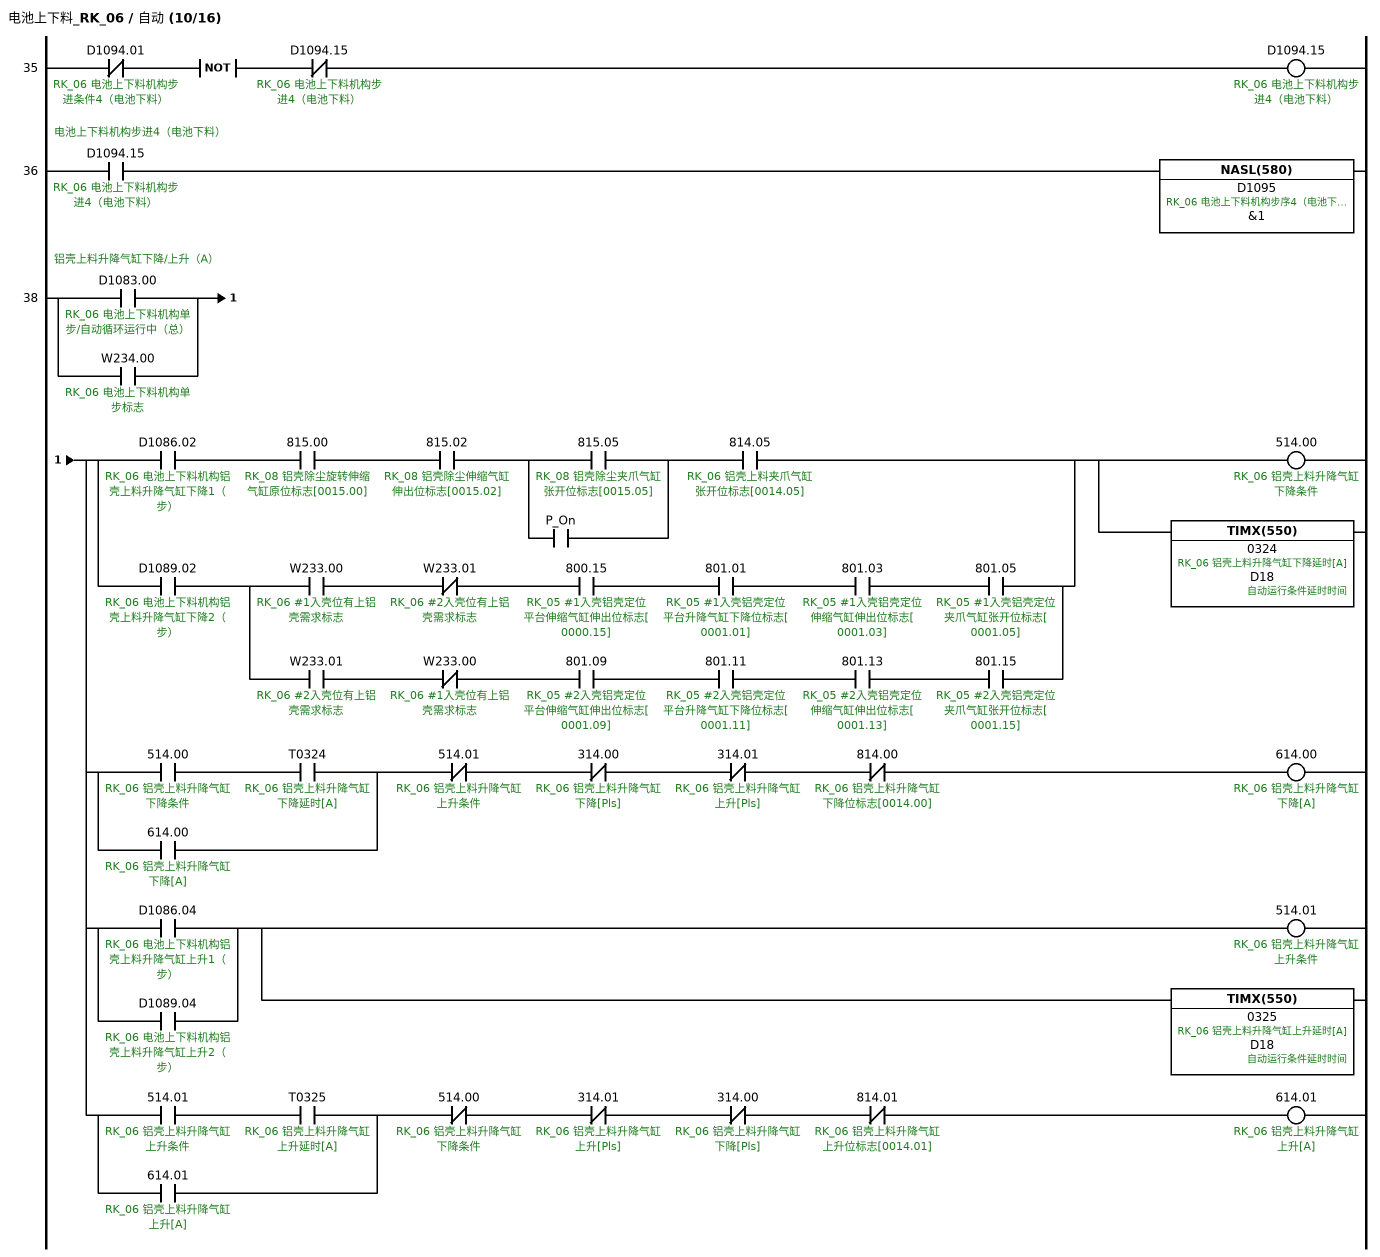
; rung 35
LDNOT D1094.01  ; RK_06 电池上下料机构步进条件4（电池下料）
NOT(520)
ANDNOT D1094.15  ; RK_06 电池上下料机构步进4（电池下料）
OUT D1094.15  ; RK_06 电池上下料机构步进4（电池下料）
; rung 36: 电池上下料机构步进4（电池下料）
LD D1094.15  ; RK_06 电池上下料机构步进4（电池下料）
NASL(580) D1095 &1  ; RK_06 电池上下料机构步序4（电池下料）
; rung 37: 电池上下料机构步序跳转4（电池下料）
; rung 38: 铝壳上料升降气缸下降/上升（A）
LD D1083.00  ; RK_06 电池上下料机构单步/自动循环运行中（总）
OR W234.00  ; RK_06 电池上下料机构单步标志
OUT TR0
LD D1086.02  ; RK_06 电池上下料机构铝壳上料升降气缸下降1（步）
AND 815.00  ; RK_08 铝壳除尘旋转伸缩气缸原位标志[0015.00]
AND 815.02  ; RK_08 铝壳除尘伸缩气缸伸出位标志[0015.02]
LD 815.05  ; RK_08 铝壳除尘夹爪气缸张开位标志[0015.05]
OR P_On
ANDLD
AND 814.05  ; RK_06 铝壳上料夹爪气缸张开位标志[0014.05]
LD D1089.02  ; RK_06 电池上下料机构铝壳上料升降气缸下降2（步）
LD W233.00  ; RK_06 #1入壳位有上铝壳需求标志
ANDNOT W233.01  ; RK_06 #2入壳位有上铝壳需求标志
AND 800.15  ; RK_05 #1入壳铝壳定位平台伸缩气缸伸出位标志[0000.15]
AND 801.01  ; RK_05 #1入壳铝壳定位平台升降气缸下降位标志[0001.01]
AND 801.03  ; RK_05 #1入壳铝壳定位伸缩气缸伸出位标志[0001.03]
AND 801.05  ; RK_05 #1入壳铝壳定位夹爪气缸张开位标志[0001.05]
LD W233.01  ; RK_06 #2入壳位有上铝壳需求标志
ANDNOT W233.00  ; RK_06 #1入壳位有上铝壳需求标志
AND 801.09  ; RK_05 #2入壳铝壳定位平台伸缩气缸伸出位标志[0001.09]
AND 801.11  ; RK_05 #2入壳铝壳定位平台升降气缸下降位标志[0001.11]
AND 801.13  ; RK_05 #2入壳铝壳定位伸缩气缸伸出位标志[0001.13]
AND 801.15  ; RK_05 #2入壳铝壳定位夹爪气缸张开位标志[0001.15]
ORLD
ANDLD
ORLD
ANDLD
OUT 514.00  ; RK_06 铝壳上料升降气缸下降条件
TIMX(550) 0324 D18  ; 自动运行条件延时时间, RK_06 铝壳上料升降气缸下降延时[A]
LD TR0
LD 514.00  ; RK_06 铝壳上料升降气缸下降条件
AND T0324  ; RK_06 铝壳上料升降气缸下降延时[A]
OR 614.00  ; RK_06 铝壳上料升降气缸下降[A]
ANDLD
ANDNOT 514.01  ; RK_06 铝壳上料升降气缸上升条件
ANDNOT 314.00  ; RK_06 铝壳上料升降气缸下降[Pls]
ANDNOT 314.01  ; RK_06 铝壳上料升降气缸上升[Pls]
ANDNOT 814.00  ; RK_06 铝壳上料升降气缸下降位标志[0014.00]
OUT 614.00  ; RK_06 铝壳上料升降气缸下降[A]
LD TR0
LD D1086.04  ; RK_06 电池上下料机构铝壳上料升降气缸上升1（步）
OR D1089.04  ; RK_06 电池上下料机构铝壳上料升降气缸上升2（步）
ANDLD
OUT 514.01  ; RK_06 铝壳上料升降气缸上升条件
TIMX(550) 0325 D18  ; 自动运行条件延时时间, RK_06 铝壳上料升降气缸上升延时[A]
LD TR0
LD 514.01  ; RK_06 铝壳上料升降气缸上升条件
AND T0325  ; RK_06 铝壳上料升降气缸上升延时[A]
OR 614.01  ; RK_06 铝壳上料升降气缸上升[A]
ANDLD
ANDNOT 514.00  ; RK_06 铝壳上料升降气缸下降条件
ANDNOT 314.01  ; RK_06 铝壳上料升降气缸上升[Pls]
ANDNOT 314.00  ; RK_06 铝壳上料升降气缸下降[Pls]
ANDNOT 814.01  ; RK_06 铝壳上料升降气缸上升位标志[0014.01]
OUT 614.01  ; RK_06 铝壳上料升降气缸上升[A]

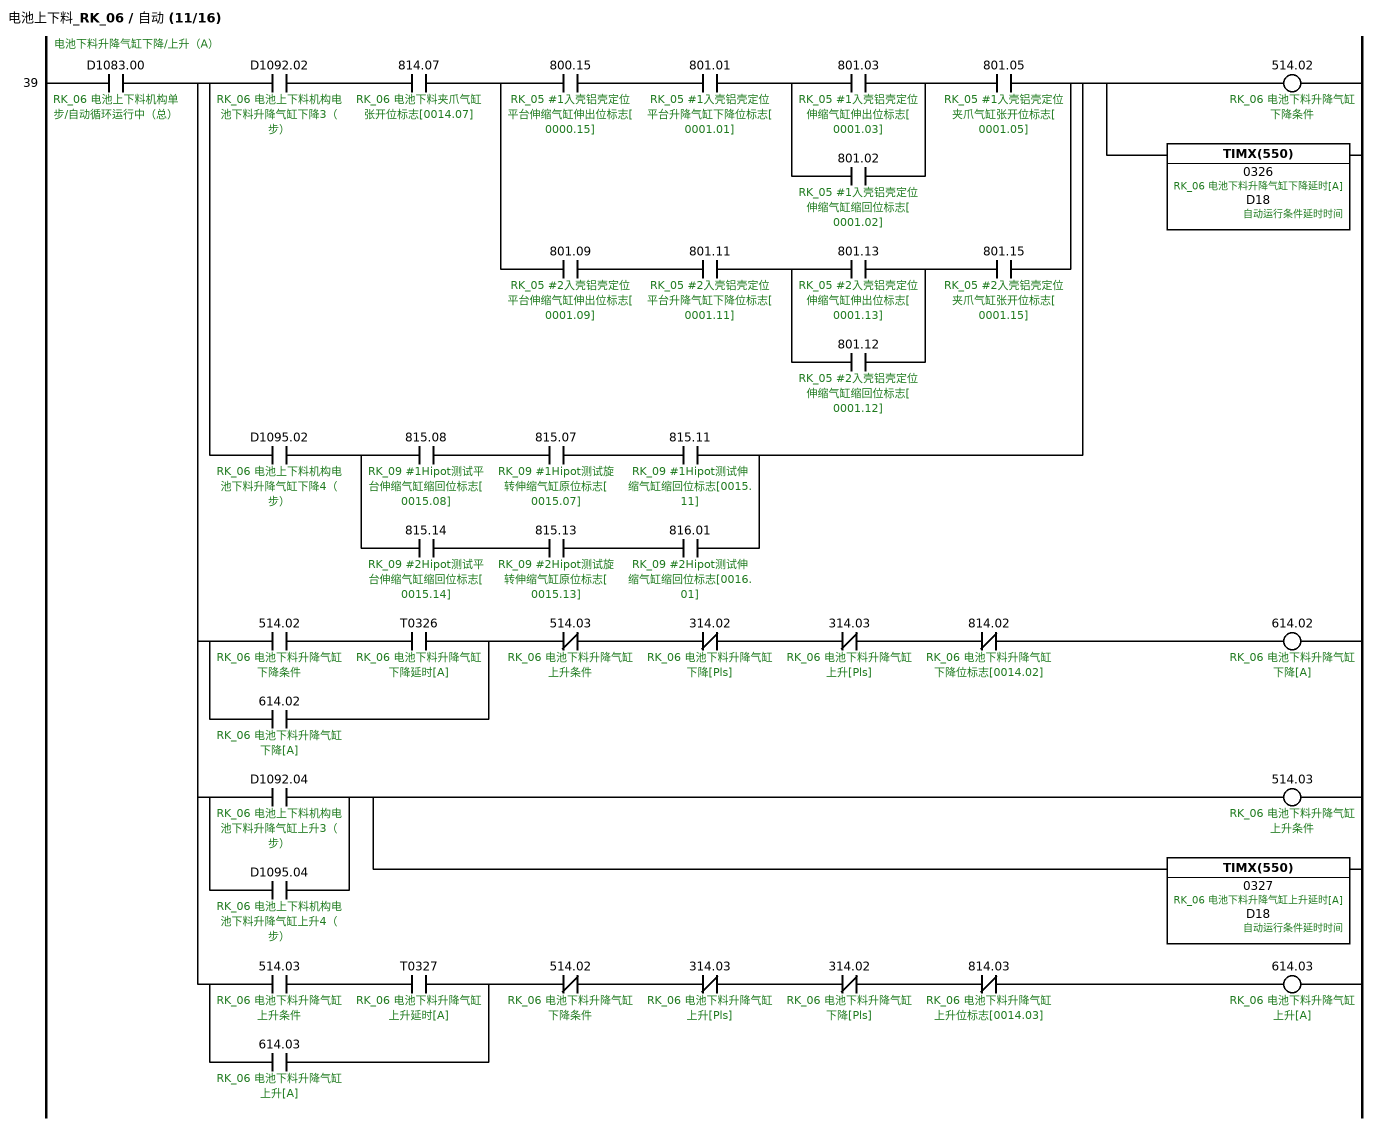
; rung 39: 电池下料升降气缸下降/上升（A）
LD D1083.00  ; RK_06 电池上下料机构单步/自动循环运行中（总）
OUT TR0
LD D1092.02  ; RK_06 电池上下料机构电池下料升降气缸下降3（步）
AND 814.07  ; RK_06 电池下料夹爪气缸张开位标志[0014.07]
LD 800.15  ; RK_05 #1入壳铝壳定位平台伸缩气缸伸出位标志[0000.15]
AND 801.01  ; RK_05 #1入壳铝壳定位平台升降气缸下降位标志[0001.01]
LD 801.03  ; RK_05 #1入壳铝壳定位伸缩气缸伸出位标志[0001.03]
OR 801.02  ; RK_05 #1入壳铝壳定位伸缩气缸缩回位标志[0001.02]
ANDLD
AND 801.05  ; RK_05 #1入壳铝壳定位夹爪气缸张开位标志[0001.05]
LD 801.09  ; RK_05 #2入壳铝壳定位平台伸缩气缸伸出位标志[0001.09]
AND 801.11  ; RK_05 #2入壳铝壳定位平台升降气缸下降位标志[0001.11]
LD 801.13  ; RK_05 #2入壳铝壳定位伸缩气缸伸出位标志[0001.13]
OR 801.12  ; RK_05 #2入壳铝壳定位伸缩气缸缩回位标志[0001.12]
ANDLD
AND 801.15  ; RK_05 #2入壳铝壳定位夹爪气缸张开位标志[0001.15]
ORLD
ANDLD
LD D1095.02  ; RK_06 电池上下料机构电池下料升降气缸下降4（步）
LD 815.08  ; RK_09 #1Hipot测试平台伸缩气缸缩回位标志[0015.08]
AND 815.07  ; RK_09 #1Hipot测试旋转伸缩气缸原位标志[0015.07]
AND 815.11  ; RK_09 #1Hipot测试伸缩气缸缩回位标志[0015.11]
LD 815.14  ; RK_09 #2Hipot测试平台伸缩气缸缩回位标志[0015.14]
AND 815.13  ; RK_09 #2Hipot测试旋转伸缩气缸原位标志[0015.13]
AND 816.01  ; RK_09 #2Hipot测试伸缩气缸缩回位标志[0016.01]
ORLD
ANDLD
ORLD
ANDLD
OUT 514.02  ; RK_06 电池下料升降气缸下降条件
TIMX(550) 0326 D18  ; 自动运行条件延时时间, RK_06 电池下料升降气缸下降延时[A]
LD TR0
LD 514.02  ; RK_06 电池下料升降气缸下降条件
AND T0326  ; RK_06 电池下料升降气缸下降延时[A]
OR 614.02  ; RK_06 电池下料升降气缸下降[A]
ANDLD
ANDNOT 514.03  ; RK_06 电池下料升降气缸上升条件
ANDNOT 314.02  ; RK_06 电池下料升降气缸下降[Pls]
ANDNOT 314.03  ; RK_06 电池下料升降气缸上升[Pls]
ANDNOT 814.02  ; RK_06 电池下料升降气缸下降位标志[0014.02]
OUT 614.02  ; RK_06 电池下料升降气缸下降[A]
LD TR0
LD D1092.04  ; RK_06 电池上下料机构电池下料升降气缸上升3（步）
OR D1095.04  ; RK_06 电池上下料机构电池下料升降气缸上升4（步）
ANDLD
OUT 514.03  ; RK_06 电池下料升降气缸上升条件
TIMX(550) 0327 D18  ; 自动运行条件延时时间, RK_06 电池下料升降气缸上升延时[A]
LD TR0
LD 514.03  ; RK_06 电池下料升降气缸上升条件
AND T0327  ; RK_06 电池下料升降气缸上升延时[A]
OR 614.03  ; RK_06 电池下料升降气缸上升[A]
ANDLD
ANDNOT 514.02  ; RK_06 电池下料升降气缸下降条件
ANDNOT 314.03  ; RK_06 电池下料升降气缸上升[Pls]
ANDNOT 314.02  ; RK_06 电池下料升降气缸下降[Pls]
ANDNOT 814.03  ; RK_06 电池下料升降气缸上升位标志[0014.03]
OUT 614.03  ; RK_06 电池下料升降气缸上升[A]

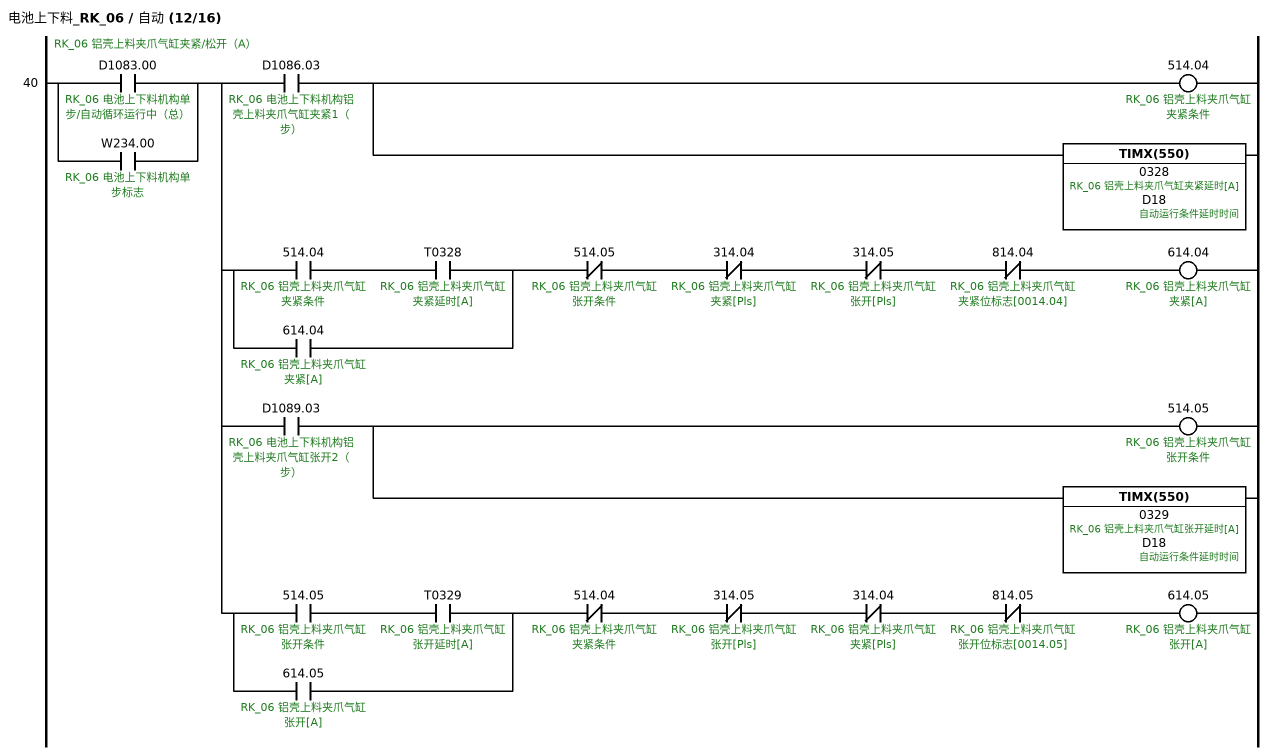
; rung 40: RK_06 铝壳上料夹爪气缸夹紧/松开（A）
LD D1083.00  ; RK_06 电池上下料机构单步/自动循环运行中（总）
OR W234.00  ; RK_06 电池上下料机构单步标志
OUT TR0
AND D1086.03  ; RK_06 电池上下料机构铝壳上料夹爪气缸夹紧1（步）
OUT 514.04  ; RK_06 铝壳上料夹爪气缸夹紧条件
TIMX(550) 0328 D18  ; 自动运行条件延时时间, RK_06 铝壳上料夹爪气缸夹紧延时[A]
LD TR0
LD 514.04  ; RK_06 铝壳上料夹爪气缸夹紧条件
AND T0328  ; RK_06 铝壳上料夹爪气缸夹紧延时[A]
OR 614.04  ; RK_06 铝壳上料夹爪气缸夹紧[A]
ANDLD
ANDNOT 514.05  ; RK_06 铝壳上料夹爪气缸张开条件
ANDNOT 314.04  ; RK_06 铝壳上料夹爪气缸夹紧[Pls]
ANDNOT 314.05  ; RK_06 铝壳上料夹爪气缸张开[Pls]
ANDNOT 814.04  ; RK_06 铝壳上料夹爪气缸夹紧位标志[0014.04]
OUT 614.04  ; RK_06 铝壳上料夹爪气缸夹紧[A]
LD TR0
AND D1089.03  ; RK_06 电池上下料机构铝壳上料夹爪气缸张开2（步）
OUT 514.05  ; RK_06 铝壳上料夹爪气缸张开条件
TIMX(550) 0329 D18  ; 自动运行条件延时时间, RK_06 铝壳上料夹爪气缸张开延时[A]
LD TR0
LD 514.05  ; RK_06 铝壳上料夹爪气缸张开条件
AND T0329  ; RK_06 铝壳上料夹爪气缸张开延时[A]
OR 614.05  ; RK_06 铝壳上料夹爪气缸张开[A]
ANDLD
ANDNOT 514.04  ; RK_06 铝壳上料夹爪气缸夹紧条件
ANDNOT 314.05  ; RK_06 铝壳上料夹爪气缸张开[Pls]
ANDNOT 314.04  ; RK_06 铝壳上料夹爪气缸夹紧[Pls]
ANDNOT 814.05  ; RK_06 铝壳上料夹爪气缸张开位标志[0014.05]
OUT 614.05  ; RK_06 铝壳上料夹爪气缸张开[A]

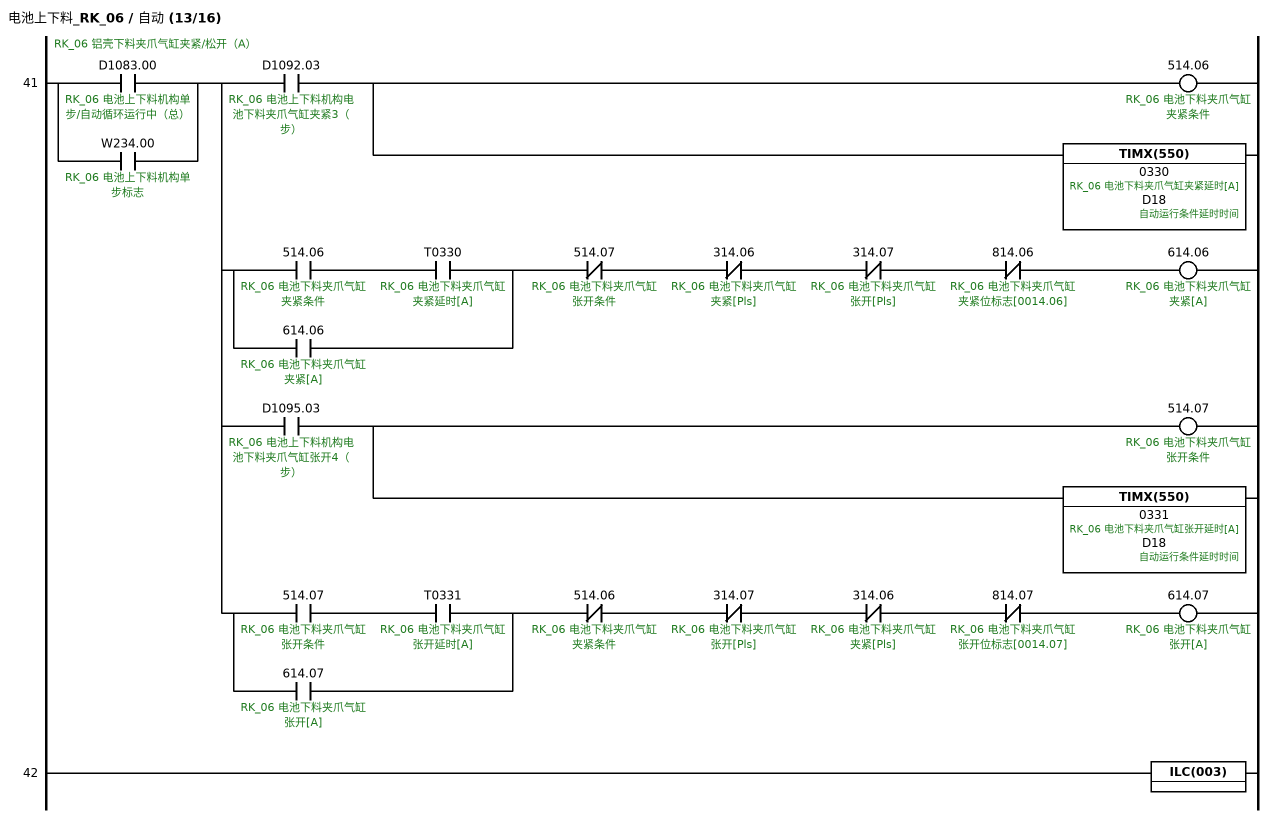
; rung 41: RK_06 铝壳下料夹爪气缸夹紧/松开（A）
LD D1083.00  ; RK_06 电池上下料机构单步/自动循环运行中（总）
OR W234.00  ; RK_06 电池上下料机构单步标志
OUT TR0
AND D1092.03  ; RK_06 电池上下料机构电池下料夹爪气缸夹紧3（步）
OUT 514.06  ; RK_06 电池下料夹爪气缸夹紧条件
TIMX(550) 0330 D18  ; 自动运行条件延时时间, RK_06 电池下料夹爪气缸夹紧延时[A]
LD TR0
LD 514.06  ; RK_06 电池下料夹爪气缸夹紧条件
AND T0330  ; RK_06 电池下料夹爪气缸夹紧延时[A]
OR 614.06  ; RK_06 电池下料夹爪气缸夹紧[A]
ANDLD
ANDNOT 514.07  ; RK_06 电池下料夹爪气缸张开条件
ANDNOT 314.06  ; RK_06 电池下料夹爪气缸夹紧[Pls]
ANDNOT 314.07  ; RK_06 电池下料夹爪气缸张开[Pls]
ANDNOT 814.06  ; RK_06 电池下料夹爪气缸夹紧位标志[0014.06]
OUT 614.06  ; RK_06 电池下料夹爪气缸夹紧[A]
LD TR0
AND D1095.03  ; RK_06 电池上下料机构电池下料夹爪气缸张开4（步）
OUT 514.07  ; RK_06 电池下料夹爪气缸张开条件
TIMX(550) 0331 D18  ; 自动运行条件延时时间, RK_06 电池下料夹爪气缸张开延时[A]
LD TR0
LD 514.07  ; RK_06 电池下料夹爪气缸张开条件
AND T0331  ; RK_06 电池下料夹爪气缸张开延时[A]
OR 614.07  ; RK_06 电池下料夹爪气缸张开[A]
ANDLD
ANDNOT 514.06  ; RK_06 电池下料夹爪气缸夹紧条件
ANDNOT 314.07  ; RK_06 电池下料夹爪气缸张开[Pls]
ANDNOT 314.06  ; RK_06 电池下料夹爪气缸夹紧[Pls]
ANDNOT 814.07  ; RK_06 电池下料夹爪气缸张开位标志[0014.07]
OUT 614.07  ; RK_06 电池下料夹爪气缸张开[A]
; rung 42
ILC(003)

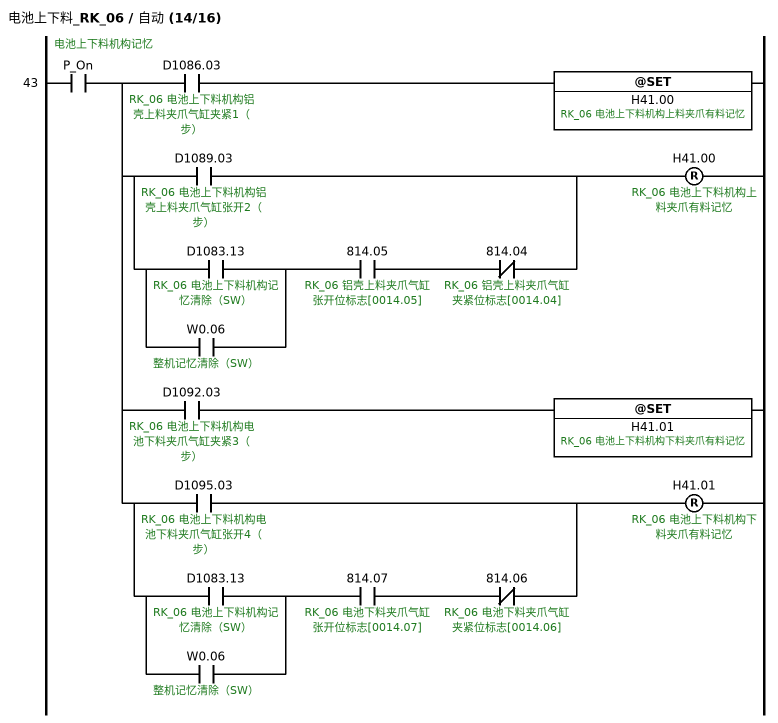
; rung 43: 电池上下料机构记忆
LD P_On
OUT TR0
AND D1086.03  ; RK_06 电池上下料机构铝壳上料夹爪气缸夹紧1（步）
@SET H41.00  ; RK_06 电池上下料机构上料夹爪有料记忆
LD TR0
LD D1089.03  ; RK_06 电池上下料机构铝壳上料夹爪气缸张开2（步）
LD D1083.13  ; RK_06 电池上下料机构记忆清除（SW）
OR W0.06  ; 整机记忆清除（SW）
AND 814.05  ; RK_06 铝壳上料夹爪气缸张开位标志[0014.05]
ANDNOT 814.04  ; RK_06 铝壳上料夹爪气缸夹紧位标志[0014.04]
ORLD
ANDLD
RSET H41.00  ; RK_06 电池上下料机构上料夹爪有料记忆
LD TR0
AND D1092.03  ; RK_06 电池上下料机构电池下料夹爪气缸夹紧3（步）
@SET H41.01  ; RK_06 电池上下料机构下料夹爪有料记忆
LD TR0
LD D1095.03  ; RK_06 电池上下料机构电池下料夹爪气缸张开4（步）
LD D1083.13  ; RK_06 电池上下料机构记忆清除（SW）
OR W0.06  ; 整机记忆清除（SW）
AND 814.07  ; RK_06 电池下料夹爪气缸张开位标志[0014.07]
ANDNOT 814.06  ; RK_06 电池下料夹爪气缸夹紧位标志[0014.06]
ORLD
ANDLD
RSET H41.01  ; RK_06 电池上下料机构下料夹爪有料记忆

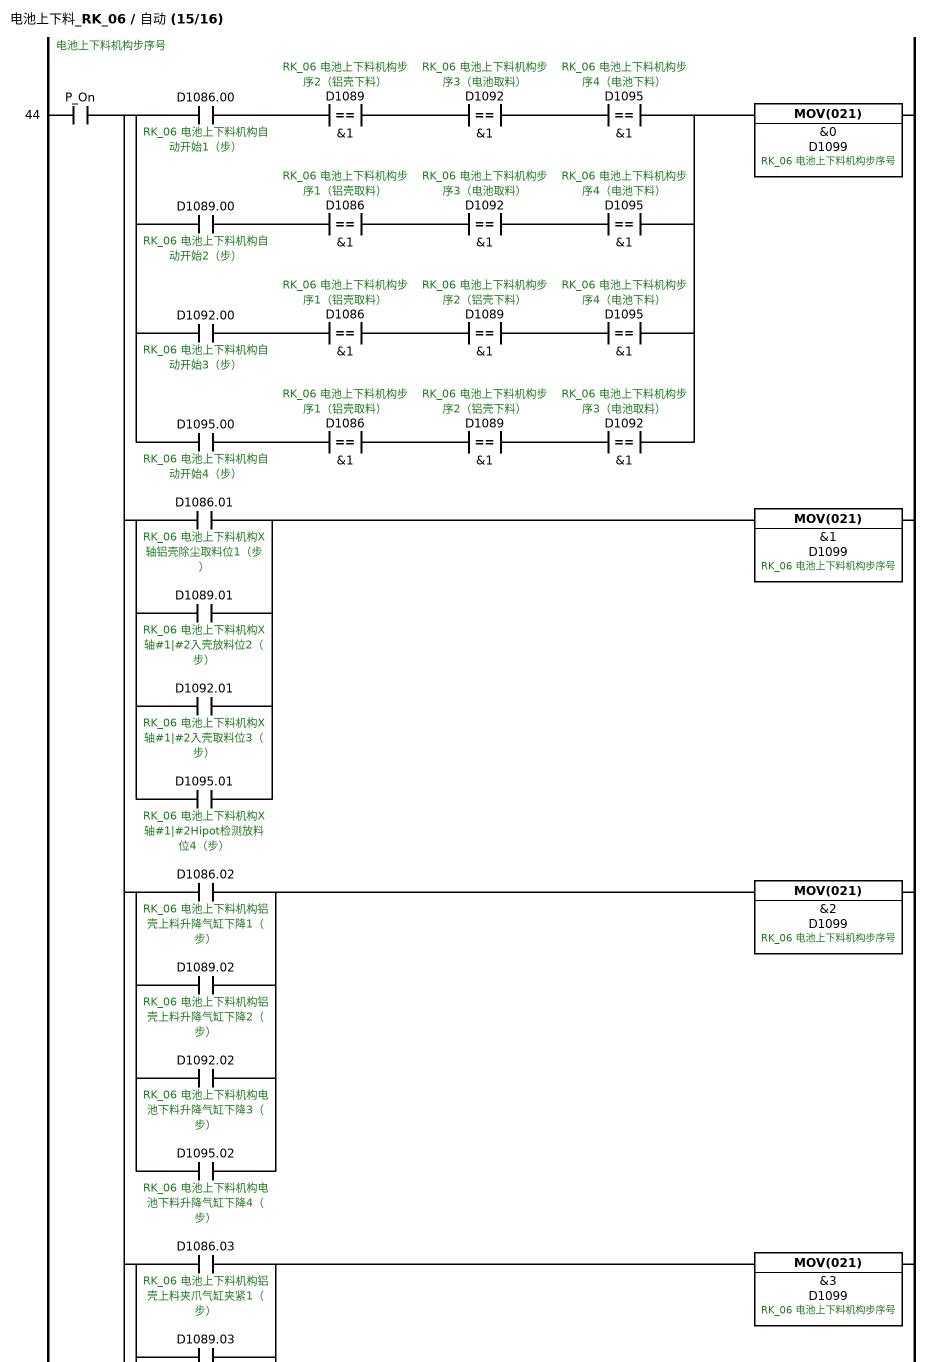

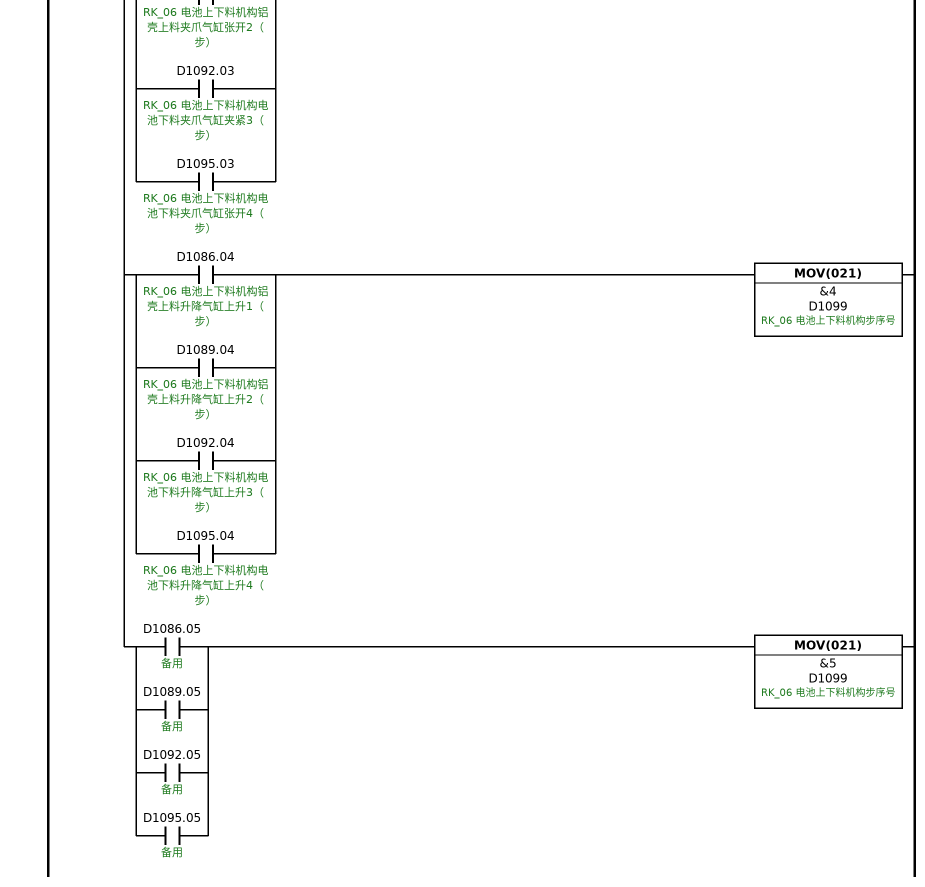
; rung 44: 电池上下料机构步序号
LD P_On
OUT TR0
LD D1086.00  ; RK_06 电池上下料机构自动开始1（步）
AND=(300) D1089 &1  ; RK_06 电池上下料机构步序2（铝壳下料）
AND=(300) D1092 &1  ; RK_06 电池上下料机构步序3（电池取料）
AND=(300) D1095 &1  ; RK_06 电池上下料机构步序4（电池下料）
LD D1089.00  ; RK_06 电池上下料机构自动开始2（步）
AND=(300) D1086 &1  ; RK_06 电池上下料机构步序1（铝壳取料）
AND=(300) D1092 &1  ; RK_06 电池上下料机构步序3（电池取料）
AND=(300) D1095 &1  ; RK_06 电池上下料机构步序4（电池下料）
ORLD
LD D1092.00  ; RK_06 电池上下料机构自动开始3（步）
AND=(300) D1086 &1  ; RK_06 电池上下料机构步序1（铝壳取料）
AND=(300) D1089 &1  ; RK_06 电池上下料机构步序2（铝壳下料）
AND=(300) D1095 &1  ; RK_06 电池上下料机构步序4（电池下料）
ORLD
LD D1095.00  ; RK_06 电池上下料机构自动开始4（步）
AND=(300) D1086 &1  ; RK_06 电池上下料机构步序1（铝壳取料）
AND=(300) D1089 &1  ; RK_06 电池上下料机构步序2（铝壳下料）
AND=(300) D1092 &1  ; RK_06 电池上下料机构步序3（电池取料）
ORLD
ANDLD
MOV(021) &0 D1099  ; RK_06 电池上下料机构步序号
LD TR0
LD D1086.01  ; RK_06 电池上下料机构X轴铝壳除尘取料位1（步）
OR D1089.01  ; RK_06 电池上下料机构X轴#1|#2入壳放料位2（步）
OR D1092.01  ; RK_06 电池上下料机构X轴#1|#2入壳取料位3（步）
OR D1095.01  ; RK_06 电池上下料机构X轴#1|#2Hipot检测放料位4（步）
ANDLD
MOV(021) &1 D1099  ; RK_06 电池上下料机构步序号
LD TR0
LD D1086.02  ; RK_06 电池上下料机构铝壳上料升降气缸下降1（步）
OR D1089.02  ; RK_06 电池上下料机构铝壳上料升降气缸下降2（步）
OR D1092.02  ; RK_06 电池上下料机构电池下料升降气缸下降3（步）
OR D1095.02  ; RK_06 电池上下料机构电池下料升降气缸下降4（步）
ANDLD
MOV(021) &2 D1099  ; RK_06 电池上下料机构步序号
LD TR0
LD D1086.03  ; RK_06 电池上下料机构铝壳上料夹爪气缸夹紧1（步）
OR D1089.03  ; RK_06 电池上下料机构铝壳上料夹爪气缸张开2（步）
OR D1092.03  ; RK_06 电池上下料机构电池下料夹爪气缸夹紧3（步）
OR D1095.03  ; RK_06 电池上下料机构电池下料夹爪气缸张开4（步）
ANDLD
MOV(021) &3 D1099  ; RK_06 电池上下料机构步序号
LD TR0
LD D1086.04  ; RK_06 电池上下料机构铝壳上料升降气缸上升1（步）
OR D1089.04  ; RK_06 电池上下料机构铝壳上料升降气缸上升2（步）
OR D1092.04  ; RK_06 电池上下料机构电池下料升降气缸上升3（步）
OR D1095.04  ; RK_06 电池上下料机构电池下料升降气缸上升4（步）
ANDLD
MOV(021) &4 D1099  ; RK_06 电池上下料机构步序号
LD TR0
LD D1086.05  ; 备用
OR D1089.05  ; 备用
OR D1092.05  ; 备用
OR D1095.05  ; 备用
ANDLD
MOV(021) &5 D1099  ; RK_06 电池上下料机构步序号

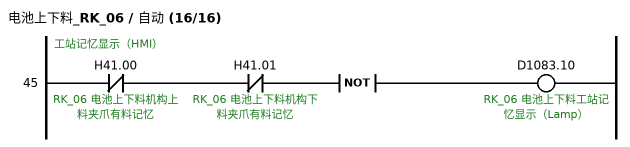
; rung 45: 工站记忆显示（HMI）
LDNOT H41.00  ; RK_06 电池上下料机构上料夹爪有料记忆
ANDNOT H41.01  ; RK_06 电池上下料机构下料夹爪有料记忆
NOT(520)
OUT D1083.10  ; RK_06 电池上下料工站记忆显示（Lamp）

### Section 复位

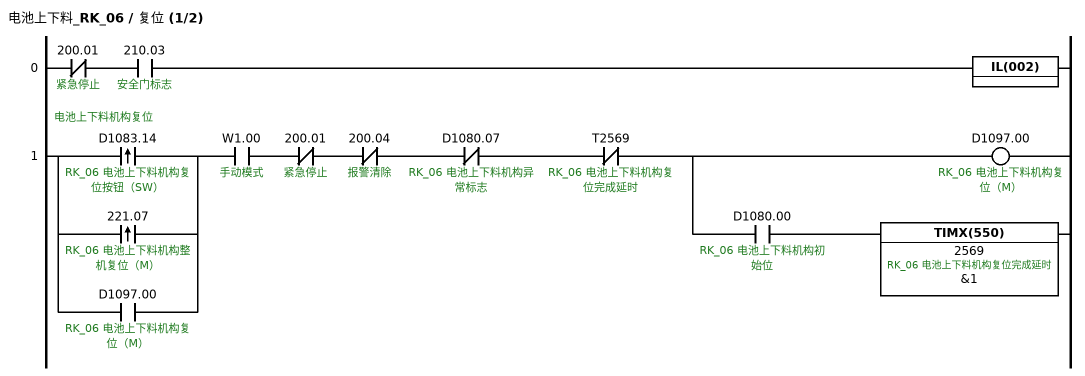
; rung 0
LDNOT 200.01  ; 紧急停止
AND 210.03  ; 安全门标志
IL(002)
; rung 1: 电池上下料机构复位
@LD D1083.14  ; RK_06 电池上下料机构复位按钮（SW）
@OR 221.07  ; RK_06 电池上下料机构整机复位（M）
OR D1097.00  ; RK_06 电池上下料机构复位（M）
AND W1.00  ; 手动模式
ANDNOT 200.01  ; 紧急停止
ANDNOT 200.04  ; 报警清除
ANDNOT D1080.07  ; RK_06 电池上下料机构异常标志
ANDNOT T2569  ; RK_06 电池上下料机构复位完成延时
OUT D1097.00  ; RK_06 电池上下料机构复位（M）
AND D1080.00  ; RK_06 电池上下料机构初始位
TIMX(550) 2569 &1  ; RK_06 电池上下料机构复位完成延时

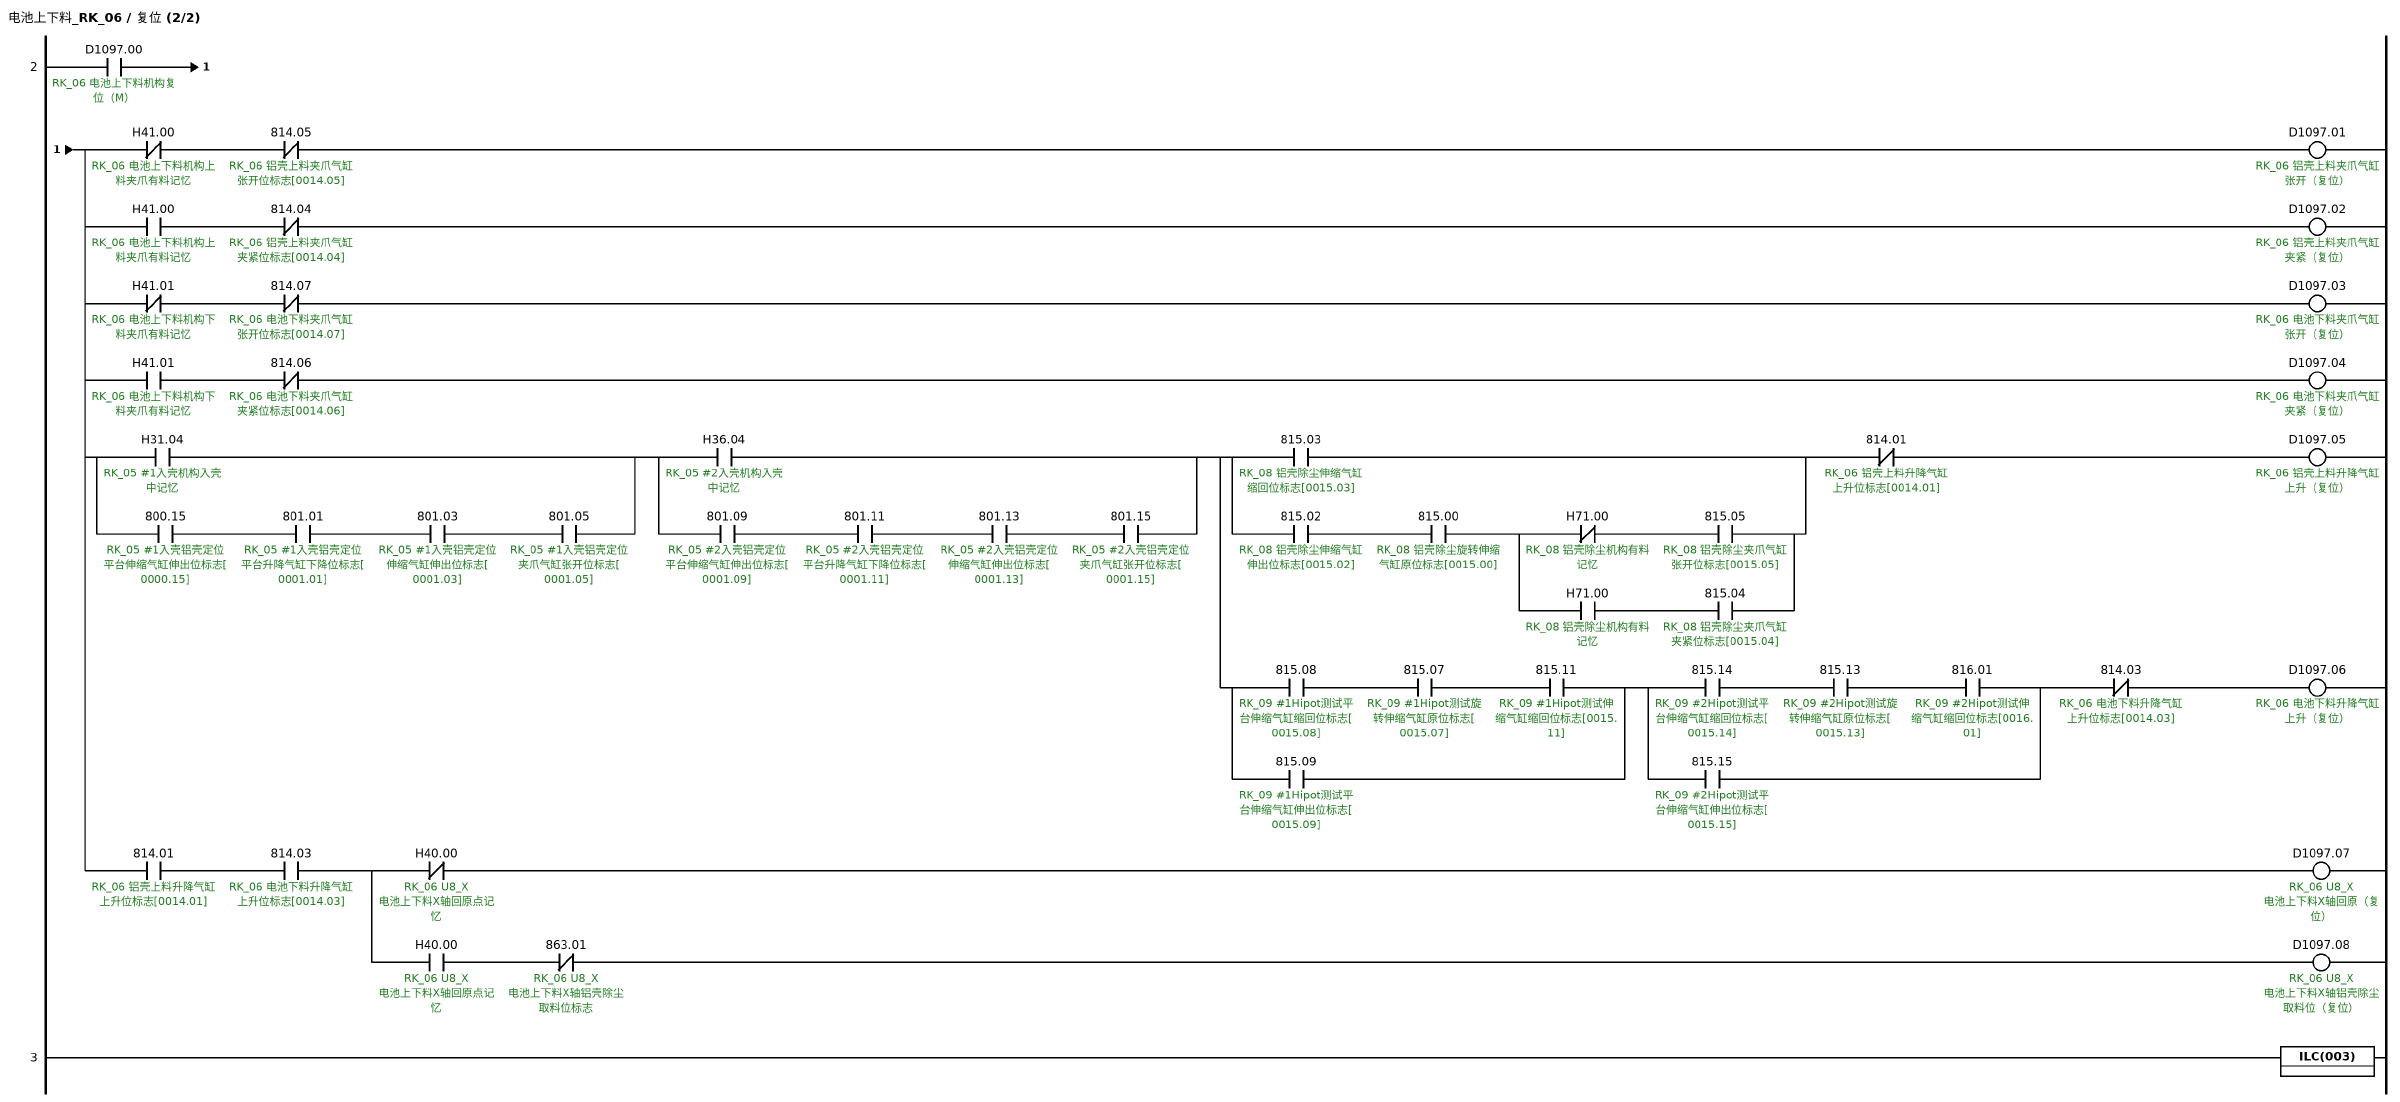
; rung 2
LD D1097.00  ; RK_06 电池上下料机构复位（M）
OUT TR0
ANDNOT H41.00  ; RK_06 电池上下料机构上料夹爪有料记忆
ANDNOT 814.05  ; RK_06 铝壳上料夹爪气缸张开位标志[0014.05]
OUT D1097.01  ; RK_06 铝壳上料夹爪气缸张开（复位）
LD TR0
AND H41.00  ; RK_06 电池上下料机构上料夹爪有料记忆
ANDNOT 814.04  ; RK_06 铝壳上料夹爪气缸夹紧位标志[0014.04]
OUT D1097.02  ; RK_06 铝壳上料夹爪气缸夹紧（复位）
LD TR0
ANDNOT H41.01  ; RK_06 电池上下料机构下料夹爪有料记忆
ANDNOT 814.07  ; RK_06 电池下料夹爪气缸张开位标志[0014.07]
OUT D1097.03  ; RK_06 电池下料夹爪气缸张开（复位）
LD TR0
AND H41.01  ; RK_06 电池上下料机构下料夹爪有料记忆
ANDNOT 814.06  ; RK_06 电池下料夹爪气缸夹紧位标志[0014.06]
OUT D1097.04  ; RK_06 电池下料夹爪气缸夹紧（复位）
LD TR0
LD H31.04  ; RK_05 #1入壳机构入壳中记忆
LD 800.15  ; RK_05 #1入壳铝壳定位平台伸缩气缸伸出位标志[0000.15]
AND 801.01  ; RK_05 #1入壳铝壳定位平台升降气缸下降位标志[0001.01]
AND 801.03  ; RK_05 #1入壳铝壳定位伸缩气缸伸出位标志[0001.03]
AND 801.05  ; RK_05 #1入壳铝壳定位夹爪气缸张开位标志[0001.05]
ORLD
ANDLD
LD H36.04  ; RK_05 #2入壳机构入壳中记忆
LD 801.09  ; RK_05 #2入壳铝壳定位平台伸缩气缸伸出位标志[0001.09]
AND 801.11  ; RK_05 #2入壳铝壳定位平台升降气缸下降位标志[0001.11]
AND 801.13  ; RK_05 #2入壳铝壳定位伸缩气缸伸出位标志[0001.13]
AND 801.15  ; RK_05 #2入壳铝壳定位夹爪气缸张开位标志[0001.15]
ORLD
ANDLD
OUT TR1
LD 815.03  ; RK_08 铝壳除尘伸缩气缸缩回位标志[0015.03]
LD 815.02  ; RK_08 铝壳除尘伸缩气缸伸出位标志[0015.02]
AND 815.00  ; RK_08 铝壳除尘旋转伸缩气缸原位标志[0015.00]
LDNOT H71.00  ; RK_08 铝壳除尘机构有料记忆
AND 815.05  ; RK_08 铝壳除尘夹爪气缸张开位标志[0015.05]
LD H71.00  ; RK_08 铝壳除尘机构有料记忆
AND 815.04  ; RK_08 铝壳除尘夹爪气缸夹紧位标志[0015.04]
ORLD
ANDLD
ORLD
ANDLD
ANDNOT 814.01  ; RK_06 铝壳上料升降气缸上升位标志[0014.01]
OUT D1097.05  ; RK_06 铝壳上料升降气缸上升（复位）
LD TR1
LD 815.08  ; RK_09 #1Hipot测试平台伸缩气缸缩回位标志[0015.08]
AND 815.07  ; RK_09 #1Hipot测试旋转伸缩气缸原位标志[0015.07]
AND 815.11  ; RK_09 #1Hipot测试伸缩气缸缩回位标志[0015.11]
OR 815.09  ; RK_09 #1Hipot测试平台伸缩气缸伸出位标志[0015.09]
ANDLD
LD 815.14  ; RK_09 #2Hipot测试平台伸缩气缸缩回位标志[0015.14]
AND 815.13  ; RK_09 #2Hipot测试旋转伸缩气缸原位标志[0015.13]
AND 816.01  ; RK_09 #2Hipot测试伸缩气缸缩回位标志[0016.01]
OR 815.15  ; RK_09 #2Hipot测试平台伸缩气缸伸出位标志[0015.15]
ANDLD
ANDNOT 814.03  ; RK_06 电池下料升降气缸上升位标志[0014.03]
OUT D1097.06  ; RK_06 电池下料升降气缸上升（复位）
LD TR0
AND 814.01  ; RK_06 铝壳上料升降气缸上升位标志[0014.01]
AND 814.03  ; RK_06 电池下料升降气缸上升位标志[0014.03]
OUT TR0
ANDNOT H40.00  ; RK_06 U8_X 电池上下料X轴回原点记忆
OUT D1097.07  ; RK_06 U8_X 电池上下料X轴回原（复位）
LD TR0
AND H40.00  ; RK_06 U8_X 电池上下料X轴回原点记忆
ANDNOT 863.01  ; RK_06 U8_X 电池上下料X轴铝壳除尘取料位标志
OUT D1097.08  ; RK_06 U8_X 电池上下料X轴铝壳除尘取料位（复位）
; rung 3
ILC(003)

### Section 指示灯

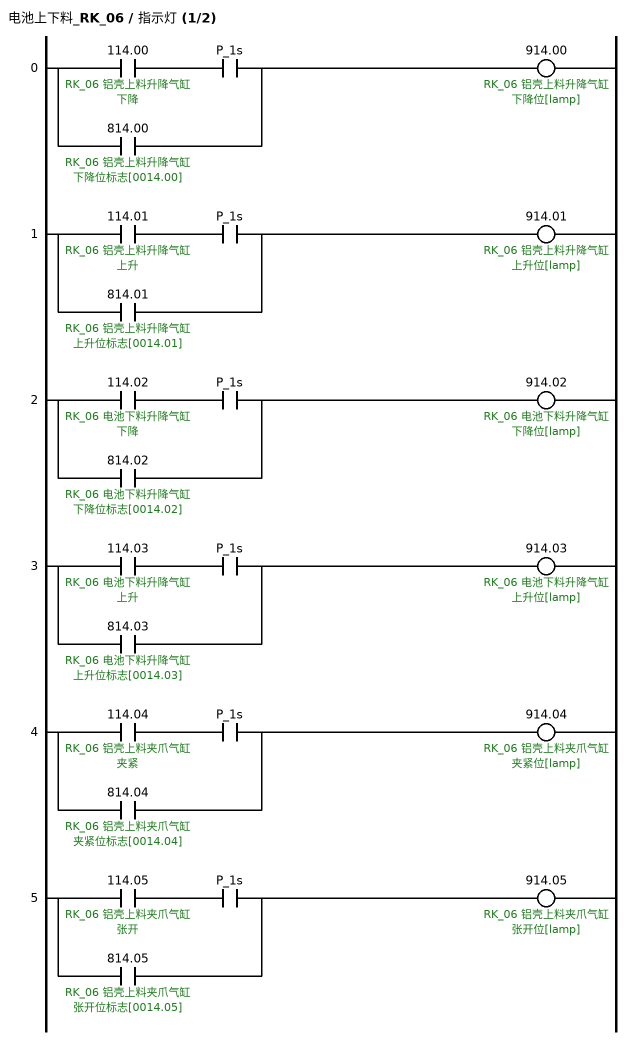
; rung 0
LD 114.00  ; RK_06 铝壳上料升降气缸下降
AND P_1s
OR 814.00  ; RK_06 铝壳上料升降气缸下降位标志[0014.00]
OUT 914.00  ; RK_06 铝壳上料升降气缸下降位[lamp]
; rung 1
LD 114.01  ; RK_06 铝壳上料升降气缸上升
AND P_1s
OR 814.01  ; RK_06 铝壳上料升降气缸上升位标志[0014.01]
OUT 914.01  ; RK_06 铝壳上料升降气缸上升位[lamp]
; rung 2
LD 114.02  ; RK_06 电池下料升降气缸下降
AND P_1s
OR 814.02  ; RK_06 电池下料升降气缸下降位标志[0014.02]
OUT 914.02  ; RK_06 电池下料升降气缸下降位[lamp]
; rung 3
LD 114.03  ; RK_06 电池下料升降气缸上升
AND P_1s
OR 814.03  ; RK_06 电池下料升降气缸上升位标志[0014.03]
OUT 914.03  ; RK_06 电池下料升降气缸上升位[lamp]
; rung 4
LD 114.04  ; RK_06 铝壳上料夹爪气缸夹紧
AND P_1s
OR 814.04  ; RK_06 铝壳上料夹爪气缸夹紧位标志[0014.04]
OUT 914.04  ; RK_06 铝壳上料夹爪气缸夹紧位[lamp]
; rung 5
LD 114.05  ; RK_06 铝壳上料夹爪气缸张开
AND P_1s
OR 814.05  ; RK_06 铝壳上料夹爪气缸张开位标志[0014.05]
OUT 914.05  ; RK_06 铝壳上料夹爪气缸张开位[lamp]

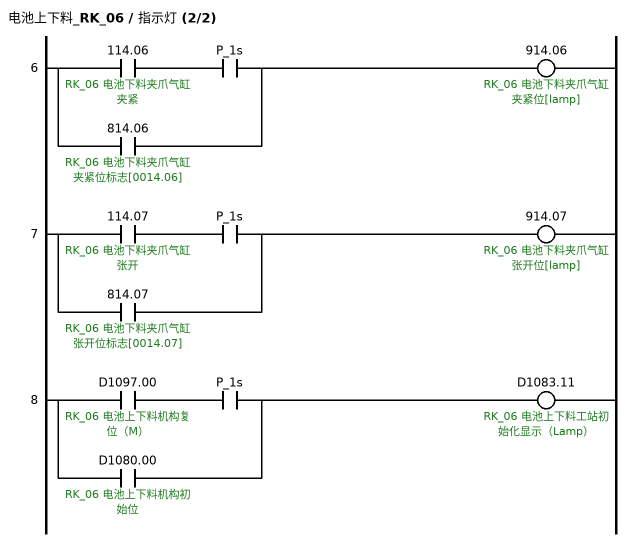
; rung 6
LD 114.06  ; RK_06 电池下料夹爪气缸夹紧
AND P_1s
OR 814.06  ; RK_06 电池下料夹爪气缸夹紧位标志[0014.06]
OUT 914.06  ; RK_06 电池下料夹爪气缸夹紧位[lamp]
; rung 7
LD 114.07  ; RK_06 电池下料夹爪气缸张开
AND P_1s
OR 814.07  ; RK_06 电池下料夹爪气缸张开位标志[0014.07]
OUT 914.07  ; RK_06 电池下料夹爪气缸张开位[lamp]
; rung 8
LD D1097.00  ; RK_06 电池上下料机构复位（M）
AND P_1s
OR D1080.00  ; RK_06 电池上下料机构初始位
OUT D1083.11  ; RK_06 电池上下料工站初始化显示（Lamp）

### Section 外部输出

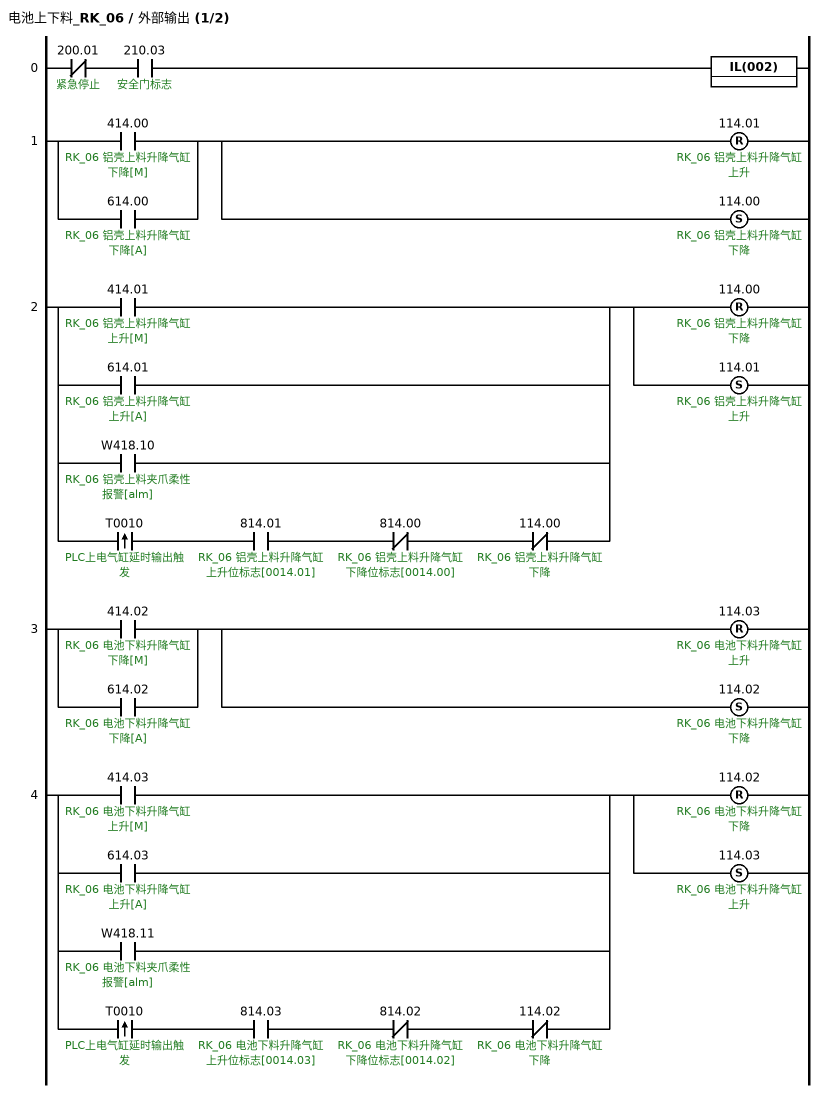
; rung 0
LDNOT 200.01  ; 紧急停止
AND 210.03  ; 安全门标志
IL(002)
; rung 1
LD 414.00  ; RK_06 铝壳上料升降气缸下降[M]
OR 614.00  ; RK_06 铝壳上料升降气缸下降[A]
RSET 114.01  ; RK_06 铝壳上料升降气缸上升
SET 114.00  ; RK_06 铝壳上料升降气缸下降
; rung 2
LD 414.01  ; RK_06 铝壳上料升降气缸上升[M]
OR 614.01  ; RK_06 铝壳上料升降气缸上升[A]
OR W418.10  ; RK_06 铝壳上料夹爪柔性报警[alm]
@LD T0010  ; PLC上电气缸延时输出触发
AND 814.01  ; RK_06 铝壳上料升降气缸上升位标志[0014.01]
ANDNOT 814.00  ; RK_06 铝壳上料升降气缸下降位标志[0014.00]
ANDNOT 114.00  ; RK_06 铝壳上料升降气缸下降
ORLD
RSET 114.00  ; RK_06 铝壳上料升降气缸下降
SET 114.01  ; RK_06 铝壳上料升降气缸上升
; rung 3
LD 414.02  ; RK_06 电池下料升降气缸下降[M]
OR 614.02  ; RK_06 电池下料升降气缸下降[A]
RSET 114.03  ; RK_06 电池下料升降气缸上升
SET 114.02  ; RK_06 电池下料升降气缸下降
; rung 4
LD 414.03  ; RK_06 电池下料升降气缸上升[M]
OR 614.03  ; RK_06 电池下料升降气缸上升[A]
OR W418.11  ; RK_06 电池下料夹爪柔性报警[alm]
@LD T0010  ; PLC上电气缸延时输出触发
AND 814.03  ; RK_06 电池下料升降气缸上升位标志[0014.03]
ANDNOT 814.02  ; RK_06 电池下料升降气缸下降位标志[0014.02]
ANDNOT 114.02  ; RK_06 电池下料升降气缸下降
ORLD
RSET 114.02  ; RK_06 电池下料升降气缸下降
SET 114.03  ; RK_06 电池下料升降气缸上升

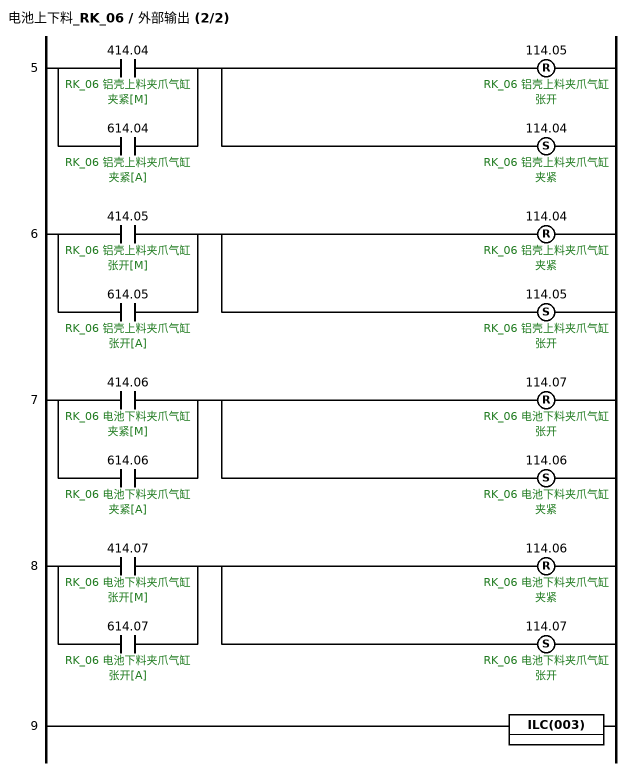
; rung 5
LD 414.04  ; RK_06 铝壳上料夹爪气缸夹紧[M]
OR 614.04  ; RK_06 铝壳上料夹爪气缸夹紧[A]
RSET 114.05  ; RK_06 铝壳上料夹爪气缸张开
SET 114.04  ; RK_06 铝壳上料夹爪气缸夹紧
; rung 6
LD 414.05  ; RK_06 铝壳上料夹爪气缸张开[M]
OR 614.05  ; RK_06 铝壳上料夹爪气缸张开[A]
RSET 114.04  ; RK_06 铝壳上料夹爪气缸夹紧
SET 114.05  ; RK_06 铝壳上料夹爪气缸张开
; rung 7
LD 414.06  ; RK_06 电池下料夹爪气缸夹紧[M]
OR 614.06  ; RK_06 电池下料夹爪气缸夹紧[A]
RSET 114.07  ; RK_06 电池下料夹爪气缸张开
SET 114.06  ; RK_06 电池下料夹爪气缸夹紧
; rung 8
LD 414.07  ; RK_06 电池下料夹爪气缸张开[M]
OR 614.07  ; RK_06 电池下料夹爪气缸张开[A]
RSET 114.06  ; RK_06 电池下料夹爪气缸夹紧
SET 114.07  ; RK_06 电池下料夹爪气缸张开
; rung 9
ILC(003)

### Section END
; rung 0
END(001)

## Program 铝壳上料（RK_07） (cyclic task 7)

### Section Main_铝壳进料

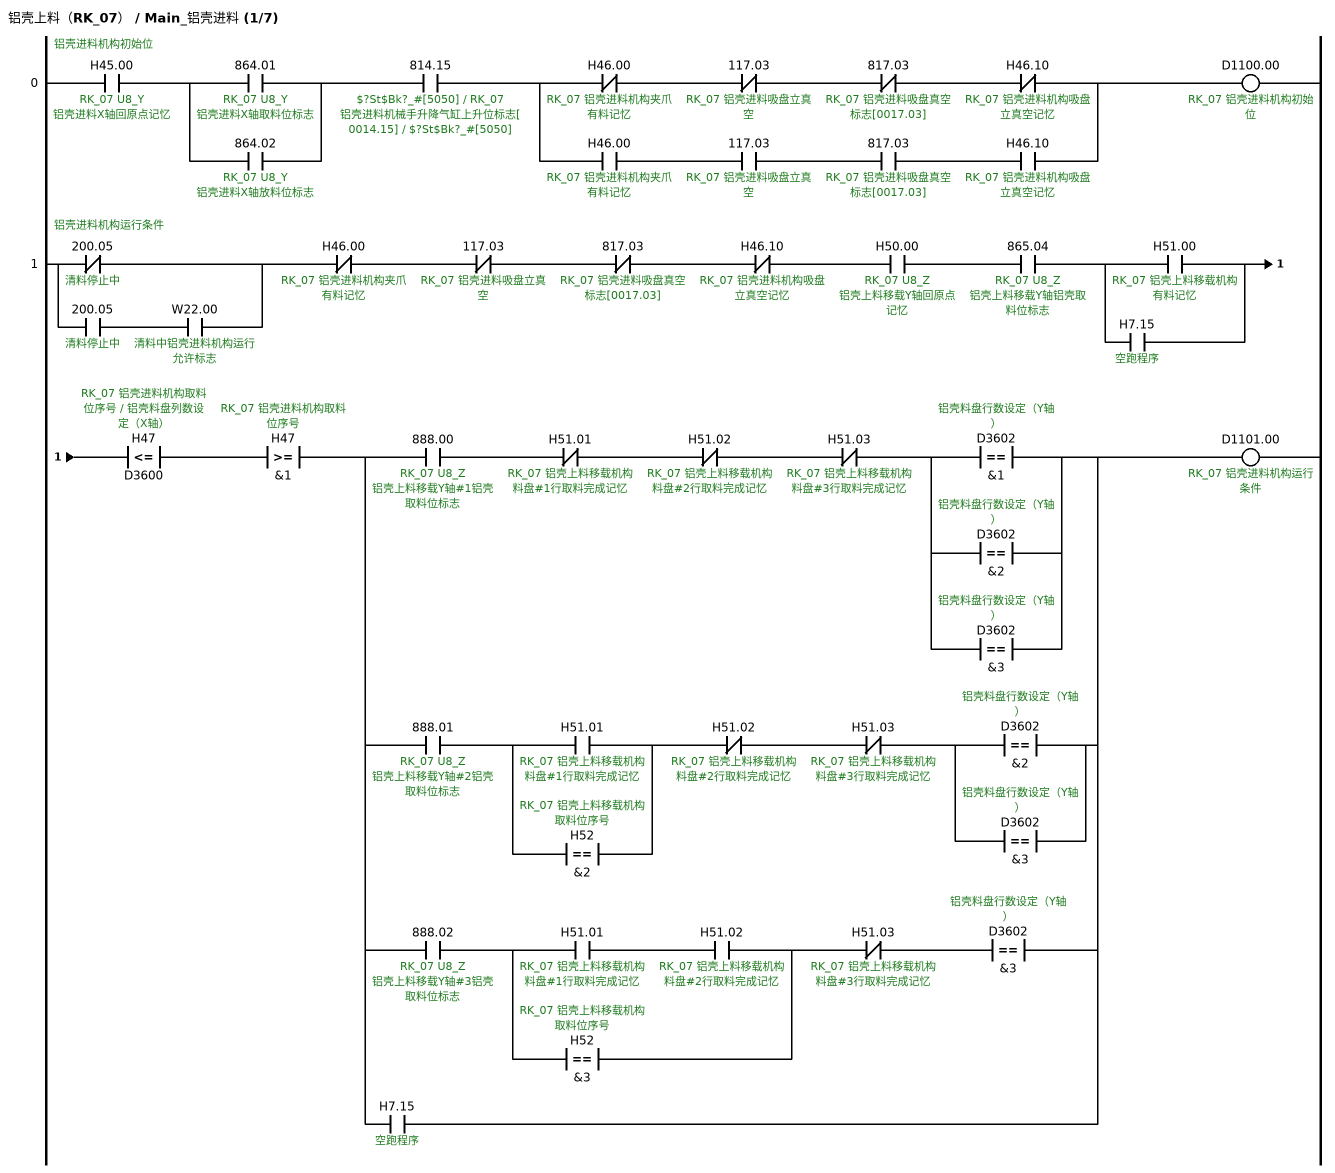
; rung 0: 铝壳进料机构初始位
LD H45.00  ; RK_07 U8_Y 铝壳进料X轴回原点记忆
LD 864.01  ; RK_07 U8_Y 铝壳进料X轴取料位标志
OR 864.02  ; RK_07 U8_Y 铝壳进料X轴放料位标志
ANDLD
AND 814.15  ; $?St$Bk?_#[5050] / RK_07 铝壳进料机械手升降气缸上升位标志[0014.15] / $?St$Bk?_#[5050]
LDNOT H46.00  ; RK_07 铝壳进料机构夹爪有料记忆
ANDNOT 117.03  ; RK_07 铝壳进料吸盘立真空
ANDNOT 817.03  ; RK_07 铝壳进料吸盘真空标志[0017.03]
ANDNOT H46.10  ; RK_07 铝壳进料机构吸盘立真空记忆
LD H46.00  ; RK_07 铝壳进料机构夹爪有料记忆
AND 117.03  ; RK_07 铝壳进料吸盘立真空
AND 817.03  ; RK_07 铝壳进料吸盘真空标志[0017.03]
AND H46.10  ; RK_07 铝壳进料机构吸盘立真空记忆
ORLD
ANDLD
OUT D1100.00  ; RK_07 铝壳进料机构初始位
; rung 1: 铝壳进料机构运行条件
LDNOT 200.05  ; 清料停止中
LD 200.05  ; 清料停止中
AND W22.00  ; 清料中铝壳进料机构运行允许标志
ORLD
ANDNOT H46.00  ; RK_07 铝壳进料机构夹爪有料记忆
ANDNOT 117.03  ; RK_07 铝壳进料吸盘立真空
ANDNOT 817.03  ; RK_07 铝壳进料吸盘真空标志[0017.03]
ANDNOT H46.10  ; RK_07 铝壳进料机构吸盘立真空记忆
AND H50.00  ; RK_07 U8_Z 铝壳上料移载Y轴回原点记忆
AND 865.04  ; RK_07 U8_Z 铝壳上料移载Y轴铝壳取料位标志
LD H51.00  ; RK_07 铝壳上料移载机构有料记忆
OR H7.15  ; 空跑程序
ANDLD
AND<=(315) H47 D3600  ; RK_07 铝壳进料机构取料位序号, 铝壳料盘列数设定（X轴）
AND>=(325) H47 &1  ; RK_07 铝壳进料机构取料位序号
LD 888.00  ; RK_07 U8_Z 铝壳上料移载Y轴#1铝壳取料位标志
ANDNOT H51.01  ; RK_07 铝壳上料移载机构料盘#1行取料完成记忆
ANDNOT H51.02  ; RK_07 铝壳上料移载机构料盘#2行取料完成记忆
ANDNOT H51.03  ; RK_07 铝壳上料移载机构料盘#3行取料完成记忆
LD=(300) D3602 &1  ; 铝壳料盘行数设定（Y轴）
OR=(300) D3602 &2  ; 铝壳料盘行数设定（Y轴）
OR=(300) D3602 &3  ; 铝壳料盘行数设定（Y轴）
ANDLD
LD 888.01  ; RK_07 U8_Z 铝壳上料移载Y轴#2铝壳取料位标志
LD H51.01  ; RK_07 铝壳上料移载机构料盘#1行取料完成记忆
OR=(300) H52 &2  ; RK_07 铝壳上料移载机构取料位序号
ANDLD
ANDNOT H51.02  ; RK_07 铝壳上料移载机构料盘#2行取料完成记忆
ANDNOT H51.03  ; RK_07 铝壳上料移载机构料盘#3行取料完成记忆
LD=(300) D3602 &2  ; 铝壳料盘行数设定（Y轴）
OR=(300) D3602 &3  ; 铝壳料盘行数设定（Y轴）
ANDLD
ORLD
LD 888.02  ; RK_07 U8_Z 铝壳上料移载Y轴#3铝壳取料位标志
LD H51.01  ; RK_07 铝壳上料移载机构料盘#1行取料完成记忆
AND H51.02  ; RK_07 铝壳上料移载机构料盘#2行取料完成记忆
OR=(300) H52 &3  ; RK_07 铝壳上料移载机构取料位序号
ANDLD
ANDNOT H51.03  ; RK_07 铝壳上料移载机构料盘#3行取料完成记忆
AND=(300) D3602 &3  ; 铝壳料盘行数设定（Y轴）
ORLD
OR H7.15  ; 空跑程序
ANDLD
OUT D1101.00  ; RK_07 铝壳进料机构运行条件

